// TwinCAT 3 PLC project SSP_M
// ProgramVersion: 3.1.4024.0
// libraries:
//   EfficientIO Communicator, * (EfficientIO)
//   EfficientIO Energy Basic, * (EfficientIO)
//   Lynus Persistent Data V1, * (Lynus AG)
//   Lynus Standards, * (EfficientIO)
//   Tc2_EtherCAT, * (Beckhoff Automation GmbH)
//   Tc2_Standard, * (Beckhoff Automation GmbH)
//   Tc2_System, * (Beckhoff Automation GmbH)
//   Tc2_Utilities, * (Beckhoff Automation GmbH)
//   Tc3_IPCDiag, * (Beckhoff Automation GmbH)
//   Tc3_Module, * (Beckhoff Automation GmbH)
// project tree:
//   ENUM/ E_State.TcDUT (not stored)
//   / FastTask.TcTTO, MiddleTask.TcTTO, SlowTask.TcTTO
//   FBs/EL3443_DPM/DUTs/ E_EL3443_DPM_Phase.TcDUT (not stored), E_EL3443_DPM_Total.TcDUT (not stored), MDP5001_341_7CD731EE.TcDUT (not stored), MDP5001_341_I_7CD731EE.TcDUT, MDP5001_341_O_7CD731EE.TcDUT (not stored), ST_EL3443_DPM_MUX_REAL.TcDUT (not stored), ST_EL3443_DPM_MUX_ULINT.TcDUT (not stored), ST_EL3443_DPM_StatusLx.TcDUT (not stored), ST_EL3443_DPM_StatusTotal.TcDUT (not stored), ST_EL3443_DPM_VariantLx.TcDUT (not stored), ST_EL3443_DPM_VariantTotal.TcDUT (not stored), ST_EL3443_DPM_VariantValues.TcDUT (not stored)
//   FBs/EL3443_DPM/ FB_EL3443_DPM.TcPOU (not stored)
//   FBs/EL3446 FW02 or higher/DUTs/ E_EL3446_Phase.TcDUT (not stored), MDP5001_342_066CA8C6.TcDUT (not stored), MDP5001_342_I_066CA8C6.TcDUT (not stored), MDP5001_342_O_066CA8C6.TcDUT (not stored), ST_EL3446_MUX_REAL.TcDUT (not stored), ST_EL3446_MUX_ULINT.TcDUT (not stored), ST_EL3446_StatusIx.TcDUT (not stored), ST_EL3446_VariantIx.TcDUT (not stored), ST_EL3446_VariantValues.TcDUT (not stored)
//   FBs/EL3446 FW02 or higher/ FB_EL3446.TcPOU (not stored)
//   FBs/ FB_CoE_EL3443.TcPOU (not stored), FB_CoE_EL3446.TcPOU (not stored), FB_EM_Beckhoff_EL3443.TcPOU (not stored), FB_EM_Beckhoff_EL3446.TcPOU (not stored), prg_ReadDeviceName.TcPOU (not stored)
//   POUs/ prgComEffIO.TcPOU, prgEM.TcPOU, prgHW.TcPOU, prgPersistent.TcPOU (not stored), prgRWEffIO.TcPOU, prgVarEffIO.TcPOU

CONFIGURATION SSP_M
    RESOURCE PLC ON TwinCAT3
        TASK FastTask(INTERVAL := T#10ms, PRIORITY := 21);
        TASK MiddleTask(INTERVAL := T#10ms, PRIORITY := 22);
        TASK SlowTask(INTERVAL := T#10ms, PRIORITY := 23);
        PROGRAM prgVarEffIO WITH FastTask : prgVarEffIO;
        PROGRAM prgRWEffIO WITH FastTask : prgRWEffIO;
        PROGRAM prgPersistent WITH MiddleTask : prgPersistent;
        PROGRAM prgEM WITH MiddleTask : prgEM;
        PROGRAM prgHW WITH MiddleTask : prgHW;
        PROGRAM prgComEffIO WITH SlowTask : prgComEffIO;
    END_RESOURCE
END_CONFIGURATION

// ---- FBs/EL3443_DPM/DUTs/MDP5001_341_I_7CD731EE.TcDUT
TYPE MDP5001_341_I_7CD731EE :
STRUCT
	MDP5001_341_L1_Status_Voltage_Sign_Bit			: BIT;
	MDP5001_341_L1_Status_Overvoltage				: BIT;
	MDP5001_341_L1_Status_Overcurrent				: BIT;
	MDP5001_341_L1_Status_Inaccurate_Voltage		: BIT;
	MDP5001_341_L1_Status_Inaccurate_Current		: BIT;
	MDP5001_341_L1_Status_Voltage_Guard_Warning		: BIT;
	MDP5001_341_L1_Status_Voltage_Guard_Error		: BIT;
	MDP5001_341_L1_Status_Current_Guard_Warning		: BIT;
	MDP5001_341_L1_Status_Current_Guard_Error		: BIT;
	MDP5001_341_L1_Status_TxPDO_Toggle				: BIT;
	MDP5001_341_L1_Basic_Voltage					: REAL;
	MDP5001_341_L1_Basic_Current					: REAL;
	MDP5001_341_L1_Power_Active_Power				: REAL;
	MDP5001_341_L1_Power_Apparent_Power				: REAL;
	MDP5001_341_L1_Power_Reactive_Power				: REAL;
	MDP5001_341_L1_Power_Power_Factor				: REAL;
	MDP5001_341_L2_Status_Voltage_Sign_Bit			: BIT;
	MDP5001_341_L2_Status_Overvoltage				: BIT;
	MDP5001_341_L2_Status_Overcurrent				: BIT;
	MDP5001_341_L2_Status_Inaccurate_Voltage		: BIT;
	MDP5001_341_L2_Status_Inaccurate_Current		: BIT;
	MDP5001_341_L2_Status_Voltage_Guard_Warning		: BIT;
	MDP5001_341_L2_Status_Voltage_Guard_Error		: BIT;
	MDP5001_341_L2_Status_Current_Guard_Warning		: BIT;
	MDP5001_341_L2_Status_Current_Guard_Error		: BIT;
	MDP5001_341_L2_Status_TxPDO_Toggle				: BIT;
	MDP5001_341_L2_Basic_Voltage					: REAL;
	MDP5001_341_L2_Basic_Current					: REAL;
	MDP5001_341_L2_Power_Active_Power				: REAL;
	MDP5001_341_L2_Power_Apparent_Power				: REAL;
	MDP5001_341_L2_Power_Reactive_Power				: REAL;
	MDP5001_341_L2_Power_Power_Factor				: REAL;
	MDP5001_341_L3_Status_Voltage_Sign_Bit			: BIT;
	MDP5001_341_L3_Status_Overvoltage				: BIT;
	MDP5001_341_L3_Status_Overcurrent				: BIT;
	MDP5001_341_L3_Status_Inaccurate_Voltage		: BIT;
	MDP5001_341_L3_Status_Inaccurate_Current		: BIT;
	MDP5001_341_L3_Status_Voltage_Guard_Warning		: BIT;
	MDP5001_341_L3_Status_Voltage_Guard_Error		: BIT;
	MDP5001_341_L3_Status_Current_Guard_Warning		: BIT;
	MDP5001_341_L3_Status_Current_Guard_Error		: BIT;
	MDP5001_341_L3_Status_TxPDO_Toggle				: BIT;
	MDP5001_341_L3_Basic_Voltage					: REAL;
	MDP5001_341_L3_Basic_Current					: REAL;
	MDP5001_341_L3_Power_Active_Power				: REAL;
	MDP5001_341_L3_Power_Apparent_Power				: REAL;
	MDP5001_341_L3_Power_Reactive_Power				: REAL;
	MDP5001_341_L3_Power_Power_Factor				: REAL;	
	MDP5001_341_Total_Status_System_State					: BIT;
	MDP5001_341_Total_Status_Grid_Direction					: BIT;
	MDP5001_341_Total_Status_Frequency_Guard_Warning		: BIT;
	MDP5001_341_Total_Status_Frequency_Guard_Error			: BIT;
	MDP5001_341_Total_Status_Neutral_Current_Guard_Warning	: BIT;
	MDP5001_341_Total_Status_Neutral_Current_Guard_Error	: BIT;
	MDP5001_341_Total_Status_Active_Power_Guard_Warning		: BIT;
	MDP5001_341_Total_Status_Active_Power_Guard_Error		: BIT;
	MDP5001_341_Total_Status_Apparent_Power_Guard_Warning	: BIT;
	MDP5001_341_Total_Status_Apparent_Power_Guard_Error		: BIT;
	MDP5001_341_Total_Status_Power_Quality_Guard_Warning	: BIT;
	MDP5001_341_Total_Status_Power_Quality_Guard_Error		: BIT;
	MDP5001_341_Total_Status_TxPDO_State					: BIT;
	MDP5001_341_Total_Status_TxPDO_Toggle					: BIT;
	MDP5001_341_Total_Status_Power_Quality_Factor			: REAL;	
	MDP5001_341_Total_Basic_Frequency						: REAL;	
	MDP5001_341_Total_Basic_Power_Factor					: REAL;	
	MDP5001_341_Total_Basic_Calculated_Neutral_Line_Current	: REAL;	
	MDP5001_341_Total_Variant_Value_In_TxPDO_Toggle			: BIT;
	MDP5001_341_Total_Variant_Value_In_Index_1_REAL			: UINT;
	MDP5001_341_Total_Variant_Value_In_Value_1_REAL			: REAL;
	MDP5001_341_Total_Variant_Value_In_Index_2_REAL			: UINT;
	MDP5001_341_Total_Variant_Value_In_Value_2_REAL			: REAL;
	MDP5001_341_Total_Variant_Value_In_Index_3_REAL			: UINT;
	MDP5001_341_Total_Variant_Value_In_Value_3_REAL			: REAL;
	MDP5001_341_Total_Variant_Value_In_Index_4_ULINT		: UINT;
	MDP5001_341_Total_Variant_Value_In_Value_4_ULINT		: ULINT;
	MDP5001_341_DPM_Data_Data_1								: UDINT;
	MDP5001_341_DPM_Data_Data_2								: UDINT;
	MDP5001_341_DPM_Data_Data_3								: UDINT;
	MDP5001_341_DPM_Data_Data_4								: UDINT;
	MDP5001_341_DPM_Data_Data_5								: UDINT;
	MDP5001_341_DPM_Data_Data_6								: UDINT;
	MDP5001_341_DPM_Data_Data_7								: UDINT;
	MDP5001_341_DPM_Data_Data_8								: UDINT;
	MDP5001_341_DPM_Data_Data_9								: UDINT;
	MDP5001_341_DPM_Data_Data_10							: UDINT;
	MDP5001_341_DPM_Data_Data_11							: UDINT;
	MDP5001_341_DPM_Data_Data_12							: UDINT;
	MDP5001_341_DPM_Data_Data_13							: UDINT;
	MDP5001_341_DPM_Data_Data_14							: UDINT;
	MDP5001_341_DPM_Data_Data_15							: UDINT;
	MDP5001_341_DPM_Data_Data_16							: UDINT;
	MDP5001_341_DPM_Data_Data_17							: UDINT;
	MDP5001_341_DPM_Data_Data_18							: UDINT;
	MDP5001_341_DPM_Data_Data_19							: UDINT;
	MDP5001_341_DPM_Data_Data_20							: UDINT;
END_STRUCT
END_TYPE

// ---- POUs/prgVarEffIO.TcPOU
PROGRAM prgVarEffIO
VAR
	fbVar		: FB_VarInfo;
END_VAR

fbVar(
	bReadInfo:= , 
	eTMCFile:= eSelectTMCFile.eDontUseTMCFile, 
	eSavePositionTMCFile:= eSavePositionOnPLC.ePostionHardDisk, 
	udiCounterFoundVariables=> , 
	bError=> , 
	bBusy=> , 
	byProgress=> , 
	udiErrorCodeOut=> , 
	eErrorVarInfo_Out=> , 
	sVarWithError=> );

END_PROGRAM

// ---- POUs/prgRWEffIO.TcPOU
PROGRAM prgRWEffIO
VAR
	fbRW1		: FB_ReadWrite_V2;
	fbRW2		: FB_ReadWrite;
	fbRW3		: FB_ReadWrite;
END_VAR

fbRW1(	eUploadType := eSelectDataUploadType.e_Change_noIntervall,
		bBusy=> , 
		bError=> , 
		udiErrorCodeOut=> , 
		eErrorReadWrite_Out=> );
		
fbRW2();
		
fbRW3();

END_PROGRAM

// ---- POUs/prgEM.TcPOU
PROGRAM prgEM
VAR
 	fb_EL3443_EM0 		: FB_EM_Beckhoff_EL3443;
	fb_EL3446_1			: FB_EM_Beckhoff_EL3446;
	fb_EL3446_2			: FB_EM_Beckhoff_EL3446;
	fb_EL3446_3			: FB_EM_Beckhoff_EL3446;
	fb_EL3446_4			: FB_EM_Beckhoff_EL3446;
	
	//EM0 (CEE32 3phase Measurement, EL3443)
	lr_RealPower_EM0		: LREAL;					//{#lynus.ag#()}
	lr_ApparentPower_EM0	: LREAL;					//{#lynus.ag#()}
	lr_ReactivePower_EM0	: LREAL;					//{#lynus.ag#()}
	lr_Frequency_EM0		: LREAL;					//{#lynus.ag#()}
	lr_Voltage_EM0_L1N		: LREAL;					//{#lynus.ag#()}
	lr_Voltage_EM0_L2N		: LREAL;					//{#lynus.ag#()}
	lr_Voltage_EM0_L3N		: LREAL;					//{#lynus.ag#()}
	lr_Voltage_EM0_L1L2		: LREAL;					//{#lynus.ag#()}
	lr_Voltage_EM0_L2L3		: LREAL;					//{#lynus.ag#()}
	lr_Voltage_EM0_L3L1		: LREAL;					//{#lynus.ag#()}
 	lr_Current_EM0_L1		: LREAL;					//{#lynus.ag#()}
	lr_Current_EM0_L2		: LREAL;					//{#lynus.ag#()}
	lr_Current_EM0_L3		: LREAL;					//{#lynus.ag#()}
	
	//EM1, EL3446-1
	lrPower_EM1_1		: LREAL;						//{#lynus.ag#()}
	lrPower_EM1_2		: LREAL;						//{#lynus.ag#()}
	lrPower_EM1_3		: LREAL;						//{#lynus.ag#()}
	lrPower_EM1_4		: LREAL;						//{#lynus.ag#()}
	lrPower_EM1_5		: LREAL;						//{#lynus.ag#()}
	lrPower_EM1_6		: LREAL;						//{#lynus.ag#()}
	lrPower_EM1_3p1		: LREAL;						//{#lynus.ag#()}
	lrPower_EM1_3p2		: LREAL;						//{#lynus.ag#()}
	
	//EM2, EL3446-2
	lrPower_EM2_1		: LREAL;						//{#lynus.ag#()}
	lrPower_EM2_2		: LREAL;						//{#lynus.ag#()}
	lrPower_EM2_3		: LREAL;						//{#lynus.ag#()}
	lrPower_EM2_4		: LREAL;						//{#lynus.ag#()}
	lrPower_EM2_5		: LREAL;						//{#lynus.ag#()}
	lrPower_EM2_6		: LREAL;						//{#lynus.ag#()}
	lrPower_EM2_3p1		: LREAL;						//{#lynus.ag#()}
	lrPower_EM2_3p2		: LREAL;						//{#lynus.ag#()}
	
	//EM3, EL3446-3
	lrPower_EM3_1		: LREAL;						//{#lynus.ag#()}
	lrPower_EM3_2		: LREAL;						//{#lynus.ag#()}
	lrPower_EM3_3		: LREAL;						//{#lynus.ag#()}
	lrPower_EM3_4		: LREAL;						//{#lynus.ag#()}
	lrPower_EM3_5		: LREAL;						//{#lynus.ag#()}
	lrPower_EM3_6		: LREAL;						//{#lynus.ag#()}
	lrPower_EM3_3p1		: LREAL;						//{#lynus.ag#()}
	lrPower_EM3_3p2		: LREAL;						//{#lynus.ag#()}
	
	//EM3, EL3446-4
	lrPower_EM4_1		: LREAL;						//{#lynus.ag#()}
	lrPower_EM4_2		: LREAL;						//{#lynus.ag#()}
	lrPower_EM4_3		: LREAL;						//{#lynus.ag#()}
	lrPower_EM4_4		: LREAL;						//{#lynus.ag#()}
	lrPower_EM4_5		: LREAL;						//{#lynus.ag#()}
	lrPower_EM4_6		: LREAL;						//{#lynus.ag#()}
	lrPower_EM4_3p1		: LREAL;						//{#lynus.ag#()}
	lrPower_EM4_3p2		: LREAL;						//{#lynus.ag#()}

END_VAR

VAR_INPUT
	stEL3443_IO_1 						: MDP5001_341_7CD731EE;
	stEL3446_IO_1 						: MDP5001_342_066CA8C6; 
	stEL3446_IO_2 						: MDP5001_342_066CA8C6;	
	stEL3446_IO_3 						: MDP5001_342_066CA8C6;	
	stEL3446_IO_4 						: MDP5001_342_066CA8C6;	
END_VAR

VAR PERSISTENT
	uiCurrentTransformerRatio_EM0	:UINT:=32;
	
	lr_EnergyCounter_EM0	: LREAL;
	lr_EnergyCounter_EM1	: LREAL;
	
	ui_PhaseSelector_EM1_1 : UINT := 1;						//{#lynus.ag#()}
	ui_PhaseSelector_EM1_2 : UINT := 2;						//{#lynus.ag#()}
	ui_PhaseSelector_EM1_3 : UINT := 3;						//{#lynus.ag#()}
	ui_PhaseSelector_EM2_1 : UINT := 1;						//{#lynus.ag#()}
	ui_PhaseSelector_EM2_2 : UINT := 2;						//{#lynus.ag#()}
	ui_PhaseSelector_EM2_3 : UINT := 3;						//{#lynus.ag#()}
	ui_PhaseSelector_EM2_4 : UINT := 1;						//{#lynus.ag#()}
	ui_PhaseSelector_EM2_5 : UINT := 2;						//{#lynus.ag#()}
	ui_PhaseSelector_EM2_6 : UINT := 3;						//{#lynus.ag#()}
	ui_PhaseSelector_EM3_1 : UINT := 1;						//{#lynus.ag#()}
	ui_PhaseSelector_EM3_2 : UINT := 2;						//{#lynus.ag#()}
	ui_PhaseSelector_EM3_3 : UINT := 3;						//{#lynus.ag#()}
	ui_PhaseSelector_EM3_4 : UINT := 1;						//{#lynus.ag#()}
	ui_PhaseSelector_EM3_5 : UINT := 2;						//{#lynus.ag#()}
	ui_PhaseSelector_EM3_6 : UINT := 3;						//{#lynus.ag#()}
	ui_PhaseSelector_EM4_1 : UINT := 1;						//{#lynus.ag#()}
	ui_PhaseSelector_EM4_2 : UINT := 2;						//{#lynus.ag#()}
	ui_PhaseSelector_EM4_3 : UINT := 3;						//{#lynus.ag#()}
	ui_PhaseSelector_EM4_4 : UINT := 1;						//{#lynus.ag#()}
	ui_PhaseSelector_EM4_5 : UINT := 2;						//{#lynus.ag#()}
	ui_PhaseSelector_EM4_6 : UINT := 3;						//{#lynus.ag#()}
	
	uiCurrentTransformerRatio_EM1_1	: UINT := 300;				//{#lynus.ag#()}
	uiCurrentTransformerRatio_EM1_2	: UINT := 300;				//{#lynus.ag#()}
	uiCurrentTransformerRatio_EM1_3	: UINT := 300;				//{#lynus.ag#()}
	uiCurrentTransformerRatio_EM2_1	: UINT := 300;				//{#lynus.ag#()}
	uiCurrentTransformerRatio_EM2_2	: UINT := 300;				//{#lynus.ag#()}
	uiCurrentTransformerRatio_EM2_3	: UINT := 300;				//{#lynus.ag#()}
	uiCurrentTransformerRatio_EM2_4	: UINT := 300;				//{#lynus.ag#()}
	uiCurrentTransformerRatio_EM2_5	: UINT := 300;				//{#lynus.ag#()}
	uiCurrentTransformerRatio_EM2_6	: UINT := 300;				//{#lynus.ag#()}
	uiCurrentTransformerRatio_EM3_1	: UINT := 300;				//{#lynus.ag#()}
	uiCurrentTransformerRatio_EM3_2	: UINT := 300;				//{#lynus.ag#()}
	uiCurrentTransformerRatio_EM3_3	: UINT := 300;				//{#lynus.ag#()}
	uiCurrentTransformerRatio_EM3_4	: UINT := 300;				//{#lynus.ag#()}
	uiCurrentTransformerRatio_EM3_5	: UINT := 300;				//{#lynus.ag#()}
	uiCurrentTransformerRatio_EM3_6	: UINT := 300;				//{#lynus.ag#()}
	uiCurrentTransformerRatio_EM4_1	: UINT := 300;				//{#lynus.ag#()}
	uiCurrentTransformerRatio_EM4_2	: UINT := 300;				//{#lynus.ag#()}
	uiCurrentTransformerRatio_EM4_3	: UINT := 300;				//{#lynus.ag#()}
	uiCurrentTransformerRatio_EM4_4	: UINT := 300;				//{#lynus.ag#()}
	uiCurrentTransformerRatio_EM4_5	: UINT := 300;				//{#lynus.ag#()}
	uiCurrentTransformerRatio_EM4_6	: UINT := 300;				//{#lynus.ag#()}
	
	b_Invers_EM1_1	:	BOOL := FALSE;							//{#lynus.ag#()}
	b_Invers_EM1_2	:	BOOL := FALSE;							//{#lynus.ag#()}
	b_Invers_EM1_3	:	BOOL := FALSE;							//{#lynus.ag#()}
	b_Invers_EM2_1	:	BOOL := FALSE;							//{#lynus.ag#()}
	b_Invers_EM2_2	:	BOOL := FALSE;							//{#lynus.ag#()}
	b_Invers_EM2_3	:	BOOL := FALSE;							//{#lynus.ag#()}
	b_Invers_EM2_4	:	BOOL := FALSE;							//{#lynus.ag#()}
	b_Invers_EM2_5	:	BOOL := FALSE;							//{#lynus.ag#()}
	b_Invers_EM2_6	:	BOOL := FALSE;							//{#lynus.ag#()}
	b_Invers_EM3_1	:	BOOL := FALSE;							//{#lynus.ag#()}
	b_Invers_EM3_2	:	BOOL := FALSE;							//{#lynus.ag#()}
	b_Invers_EM3_3	:	BOOL := FALSE;							//{#lynus.ag#()}
	b_Invers_EM3_4	:	BOOL := FALSE;							//{#lynus.ag#()}
	b_Invers_EM3_5	:	BOOL := FALSE;							//{#lynus.ag#()}
	b_Invers_EM3_6	:	BOOL := FALSE;							//{#lynus.ag#()}
	b_Invers_EM4_1	:	BOOL := FALSE;							//{#lynus.ag#()}
	b_Invers_EM4_2	:	BOOL := FALSE;							//{#lynus.ag#()}
	b_Invers_EM4_3	:	BOOL := FALSE;							//{#lynus.ag#()}
	b_Invers_EM4_4	:	BOOL := FALSE;							//{#lynus.ag#()}
	b_Invers_EM4_5	:	BOOL := FALSE;							//{#lynus.ag#()}
	b_Invers_EM4_6	:	BOOL := FALSE;							//{#lynus.ag#()}
END_VAR

//EM0 (CEE32 3phase Measurement)
fb_EL3443_EM0(
	bEnable 	:= TRUE, 
	bInvers_CH1 := , 
	bInvers_CH2	:= , 
	bInvers_CH3	:= , 
	uiCurrentTransformerRatio:= uiCurrentTransformerRatio_EM0, 
	nSlaveAddr 	:= 1001,
	stEL3443_IO := ,
	pDpmData=> , 
	stDataEMPower=> , 
	stDataEMCounter=> , 
	stDataEMPowerRealTime=> , 
	stDataEMCounterRealTime=> );

fb_EL3443_EM0.stEL3443_IO.MDP5001_341_Input := stEL3443_IO_1.MDP5001_341_Input;
stEL3443_IO_1.MDP5001_341_Output	:= fb_EL3443_EM0.stEL3443_IO.MDP5001_341_Output;
 	
lr_RealPower_EM0 			:= fb_EL3443_EM0.stDataEMPower.lrPowerTotal; 	
lr_ApparentPower_EM0 		:= fb_EL3443_EM0.stDataEMPower.lrApparentPowerTotal;
lr_ReactivePower_EM0		:= fb_EL3443_EM0.stDataEMPower.lrReactivePowerTotal;
lr_Frequency_EM0			:= fb_EL3443_EM0.stDataEMPower.lrFrequency;
lr_Voltage_EM0_L1N			:= fb_EL3443_EM0.stDataEMPower.lrVoltageL1N;
lr_Voltage_EM0_L2N			:= fb_EL3443_EM0.stDataEMPower.lrVoltageL2N;
lr_Voltage_EM0_L3N			:= fb_EL3443_EM0.stDataEMPower.lrVoltageL3N;
lr_Voltage_EM0_L1L2			:= fb_EL3443_EM0.stDataEMPower.lrVoltageL1L2;
lr_Voltage_EM0_L2L3			:= fb_EL3443_EM0.stDataEMPower.lrVoltageL2L3;
lr_Voltage_EM0_L3L1			:= fb_EL3443_EM0.stDataEMPower.lrVoltageL3L1;
lr_EnergyCounter_EM0		:= fb_EL3443_EM0.stDataEMCounter.lrTotalCounterEnergy_Consumption;
lr_Current_EM0_L1			:= fb_EL3443_EM0.stDataEMPower.lrCurrentL1;
lr_Current_EM0_L2			:= fb_EL3443_EM0.stDataEMPower.lrCurrentL2;
lr_Current_EM0_L3			:= fb_EL3443_EM0.stDataEMPower.lrCurrentL3;


//EM1 (for single Phase Measurements, EL3446-1)
fb_EL3446_1(
	bEnable:= TRUE , 
	bEnableVariantValues:= TRUE, 
	pDpmData:= fb_EL3443_EM0.pDpmData, 
	nSlaveAddr:= 1002, 
	bInvers_CH1:= b_Invers_EM2_1, 
	bInvers_CH2:= b_Invers_EM2_2, 
	bInvers_CH3:= b_Invers_EM2_3, 
	bInvers_CH4:= b_Invers_EM2_4, 
	bInvers_CH5:= b_Invers_EM2_5, 
	bInvers_CH6:= b_Invers_EM2_6, 
	uiCurrentTransformerRatio_CH1:= uiCurrentTransformerRatio_EM2_1, 
	uiCurrentTransformerRatio_CH2:= uiCurrentTransformerRatio_EM2_2, 
	uiCurrentTransformerRatio_CH3:= uiCurrentTransformerRatio_EM2_3, 
	uiCurrentTransformerRatio_CH4:= uiCurrentTransformerRatio_EM2_4, 
	uiCurrentTransformerRatio_CH5:= uiCurrentTransformerRatio_EM2_5, 
	uiCurrentTransformerRatio_CH6:= uiCurrentTransformerRatio_EM2_6, 
	uiVoltagePhaseSelector_CH1:= ui_PhaseSelector_EM2_1, 
	uiVoltagePhaseSelector_CH2:= ui_PhaseSelector_EM2_2, 
	uiVoltagePhaseSelector_CH3:= ui_PhaseSelector_EM2_3, 
	uiVoltagePhaseSelector_CH4:= ui_PhaseSelector_EM2_4, 
	uiVoltagePhaseSelector_CH5:= ui_PhaseSelector_EM2_5, 
	uiVoltagePhaseSelector_CH6:= ui_PhaseSelector_EM2_6, 
	bEnable3PhaseCH13:= FALSE, 
	bEnable3PhaseCH46:= FALSE, 
	stDataEMPowerRealTime:= fb_EL3443_EM0.stDataEMPowerRealTime, 
	stEL3446_IO := ,
	stDataEMPower_CH1=> , 
	stDataEMCounter_CH1=> , 
	stDataEMPowerRealTime_CH1=> , 
	stDataEMCounterRealTime_CH1=> , 
	stDataEMPower_CH2=> , 
	stDataEMCounter_CH2=> , 
	stDataEMPowerRealTime_CH2=> , 
	stDataEMCounterRealTime_CH2=> , 
	stDataEMPower_CH3=> , 
	stDataEMCounter_CH3=> , 
	stDataEMPowerRealTime_CH3=> , 
	stDataEMCounterRealTime_CH3=> , 
	stDataEMPower_CH4=> , 
	stDataEMCounter_CH4=> , 
	stDataEMPowerRealTime_CH4=> , 
	stDataEMCounterRealTime_CH4=> , 
	stDataEMPower_CH5=> , 
	stDataEMCounter_CH5=> , 
	stDataEMPowerRealTime_CH5=> , 
	stDataEMCounterRealTime_CH5=> , 
	stDataEMPower_CH6=> , 
	stDataEMCounter_CH6=> , 
	stDataEMPowerRealTime_CH6=> , 
	stDataEMCounterRealTime_CH6=> );
fb_EL3446_1.stEL3446_IO.MDP5001_342_Input := stEL3446_IO_1.MDP5001_342_Input;
stEL3446_IO_1.MDP5001_342_Output := 	fb_EL3446_1.stEL3446_IO.MDP5001_342_Output;

lrPower_EM2_1				:= 	LIMIT(0,fb_EL3446_1.stDataEMPower_CH1.lrPowerTotal,1000);
lrPower_EM2_2				:= 	LIMIT(0,fb_EL3446_1.stDataEMPower_CH2.lrPowerTotal,1000);
lrPower_EM2_3				:= 	LIMIT(0,fb_EL3446_1.stDataEMPower_CH3.lrPowerTotal,1000);
lrPower_EM2_4				:= 	LIMIT(0,fb_EL3446_1.stDataEMPower_CH4.lrPowerTotal,1000);
lrPower_EM2_5				:= 	LIMIT(0,fb_EL3446_1.stDataEMPower_CH5.lrPowerTotal,1000);
lrPower_EM2_6				:= 	LIMIT(0,fb_EL3446_1.stDataEMPower_CH6.lrPowerTotal,1000);

lrPower_EM2_3p1 			:= lrPower_EM2_1 + lrPower_EM2_2 + lrPower_EM2_3;
lrPower_EM2_3p2 			:= lrPower_EM2_4 + lrPower_EM2_5 + lrPower_EM2_6;

//EM2 (for single Phase Measurements, EL3446-2)
fb_EL3446_2(
	bEnable:= TRUE , 
	bEnableVariantValues:= TRUE, 
	pDpmData:= fb_EL3443_EM0.pDpmData, 
	nSlaveAddr:= 1003, 
	bInvers_CH1:= b_Invers_EM2_1, 
	bInvers_CH2:= b_Invers_EM2_2, 
	bInvers_CH3:= b_Invers_EM2_3, 
	bInvers_CH4:= b_Invers_EM2_4, 
	bInvers_CH5:= b_Invers_EM2_5, 
	bInvers_CH6:= b_Invers_EM2_6, 
	uiCurrentTransformerRatio_CH1:= uiCurrentTransformerRatio_EM2_1, 
	uiCurrentTransformerRatio_CH2:= uiCurrentTransformerRatio_EM2_2, 
	uiCurrentTransformerRatio_CH3:= uiCurrentTransformerRatio_EM2_3, 
	uiCurrentTransformerRatio_CH4:= uiCurrentTransformerRatio_EM2_4, 
	uiCurrentTransformerRatio_CH5:= uiCurrentTransformerRatio_EM2_5, 
	uiCurrentTransformerRatio_CH6:= uiCurrentTransformerRatio_EM2_6, 
	uiVoltagePhaseSelector_CH1:= ui_PhaseSelector_EM2_1, 
	uiVoltagePhaseSelector_CH2:= ui_PhaseSelector_EM2_2, 
	uiVoltagePhaseSelector_CH3:= ui_PhaseSelector_EM2_3, 
	uiVoltagePhaseSelector_CH4:= ui_PhaseSelector_EM2_4, 
	uiVoltagePhaseSelector_CH5:= ui_PhaseSelector_EM2_5, 
	uiVoltagePhaseSelector_CH6:= ui_PhaseSelector_EM2_6, 
	bEnable3PhaseCH13:= FALSE, 
	bEnable3PhaseCH46:= FALSE, 
	stDataEMPowerRealTime:= fb_EL3443_EM0.stDataEMPowerRealTime, 
	stEL3446_IO := ,
	stDataEMPower_CH1=> , 
	stDataEMCounter_CH1=> , 
	stDataEMPowerRealTime_CH1=> , 
	stDataEMCounterRealTime_CH1=> , 
	stDataEMPower_CH2=> , 
	stDataEMCounter_CH2=> , 
	stDataEMPowerRealTime_CH2=> , 
	stDataEMCounterRealTime_CH2=> , 
	stDataEMPower_CH3=> , 
	stDataEMCounter_CH3=> , 
	stDataEMPowerRealTime_CH3=> , 
	stDataEMCounterRealTime_CH3=> , 
	stDataEMPower_CH4=> , 
	stDataEMCounter_CH4=> , 
	stDataEMPowerRealTime_CH4=> , 
	stDataEMCounterRealTime_CH4=> , 
	stDataEMPower_CH5=> , 
	stDataEMCounter_CH5=> , 
	stDataEMPowerRealTime_CH5=> , 
	stDataEMCounterRealTime_CH5=> , 
	stDataEMPower_CH6=> , 
	stDataEMCounter_CH6=> , 
	stDataEMPowerRealTime_CH6=> , 
	stDataEMCounterRealTime_CH6=> );
fb_EL3446_1.stEL3446_IO.MDP5001_342_Input := stEL3446_IO_1.MDP5001_342_Input;
stEL3446_IO_1.MDP5001_342_Output := 	fb_EL3446_1.stEL3446_IO.MDP5001_342_Output;

lrPower_EM2_1				:= 	LIMIT(0,fb_EL3446_1.stDataEMPower_CH1.lrPowerTotal,1000);
lrPower_EM2_2				:= 	LIMIT(0,fb_EL3446_1.stDataEMPower_CH2.lrPowerTotal,1000);
lrPower_EM2_3				:= 	LIMIT(0,fb_EL3446_1.stDataEMPower_CH3.lrPowerTotal,1000);
lrPower_EM2_4				:= 	LIMIT(0,fb_EL3446_1.stDataEMPower_CH4.lrPowerTotal,1000);
lrPower_EM2_5				:= 	LIMIT(0,fb_EL3446_1.stDataEMPower_CH5.lrPowerTotal,1000);
lrPower_EM2_6				:= 	LIMIT(0,fb_EL3446_1.stDataEMPower_CH6.lrPowerTotal,1000);

lrPower_EM2_3p1 			:= lrPower_EM2_1 + lrPower_EM2_2 + lrPower_EM2_3;
lrPower_EM2_3p2 			:= lrPower_EM2_4 + lrPower_EM2_5 + lrPower_EM2_6;

(*
lr_EnergyCounter_EM1	:= 	fb_EL3446_1.stDataEMCounter_CH1.lrTotalCounterEnergy_Consumption;
lr_EnergyCounter_EM2	:= 	fb_EL3446_1.stDataEMCounter_CH2.lrTotalCounterEnergy_Consumption;
lr_EnergyCounter_EM3	:= 	fb_EL3446_1.stDataEMCounter_CH3.lrTotalCounterEnergy_Consumption;
lr_EnergyCounter_EM4	:= 	fb_EL3446_1.stDataEMCounter_CH4.lrTotalCounterEnergy_Consumption;
lr_EnergyCounter_EM5	:= 	fb_EL3446_1.stDataEMCounter_CH5.lrTotalCounterEnergy_Consumption;
lr_EnergyCounter_EM6	:= 	fb_EL3446_1.stDataEMCounter_CH6.lrTotalCounterEnergy_Consumption;
*)

//EM3 (for single Phase Measurements, EL3446-3)
fb_EL3446_3(
	bEnable:= TRUE , 
	bEnableVariantValues:= TRUE, 
	pDpmData:= fb_EL3443_EM0.pDpmData, 
	nSlaveAddr:= 1004, 
	bInvers_CH1:= b_Invers_EM3_1, 
	bInvers_CH2:= b_Invers_EM3_2, 
	bInvers_CH3:= b_Invers_EM3_3, 
	bInvers_CH4:= b_Invers_EM3_4, 
	bInvers_CH5:= b_Invers_EM3_5, 
	bInvers_CH6:= b_Invers_EM3_6, 
	uiCurrentTransformerRatio_CH1:= uiCurrentTransformerRatio_EM3_1, 
	uiCurrentTransformerRatio_CH2:= uiCurrentTransformerRatio_EM3_2, 
	uiCurrentTransformerRatio_CH3:= uiCurrentTransformerRatio_EM3_3, 
	uiCurrentTransformerRatio_CH4:= uiCurrentTransformerRatio_EM3_4, 
	uiCurrentTransformerRatio_CH5:= uiCurrentTransformerRatio_EM3_5, 
	uiCurrentTransformerRatio_CH6:= uiCurrentTransformerRatio_EM3_6, 
	uiVoltagePhaseSelector_CH1:= ui_PhaseSelector_EM3_1, 
	uiVoltagePhaseSelector_CH2:= ui_PhaseSelector_EM3_2, 
	uiVoltagePhaseSelector_CH3:= ui_PhaseSelector_EM3_3, 
	uiVoltagePhaseSelector_CH4:= ui_PhaseSelector_EM3_4, 
	uiVoltagePhaseSelector_CH5:= ui_PhaseSelector_EM3_5, 
	uiVoltagePhaseSelector_CH6:= ui_PhaseSelector_EM3_6, 
	bEnable3PhaseCH13:= FALSE, 
	bEnable3PhaseCH46:= FALSE, 
	stDataEMPowerRealTime:= fb_EL3443_EM0.stDataEMPowerRealTime, 
	stEL3446_IO := ,
	stDataEMPower_CH1=> , 
	stDataEMCounter_CH1=> , 
	stDataEMPowerRealTime_CH1=> , 
	stDataEMCounterRealTime_CH1=> , 
	stDataEMPower_CH2=> , 
	stDataEMCounter_CH2=> , 
	stDataEMPowerRealTime_CH2=> , 
	stDataEMCounterRealTime_CH2=> , 
	stDataEMPower_CH3=> , 
	stDataEMCounter_CH3=> , 
	stDataEMPowerRealTime_CH3=> , 
	stDataEMCounterRealTime_CH3=> , 
	stDataEMPower_CH4=> , 
	stDataEMCounter_CH4=> , 
	stDataEMPowerRealTime_CH4=> , 
	stDataEMCounterRealTime_CH4=> , 
	stDataEMPower_CH5=> , 
	stDataEMCounter_CH5=> , 
	stDataEMPowerRealTime_CH5=> , 
	stDataEMCounterRealTime_CH5=> , 
	stDataEMPower_CH6=> , 
	stDataEMCounter_CH6=> , 
	stDataEMPowerRealTime_CH6=> , 
	stDataEMCounterRealTime_CH6=> );
fb_EL3446_2.stEL3446_IO.MDP5001_342_Input := stEL3446_IO_2.MDP5001_342_Input;
stEL3446_IO_2.MDP5001_342_Output := 	fb_EL3446_2.stEL3446_IO.MDP5001_342_Output;

lrPower_EM3_1				:= 	LIMIT(0,fb_EL3446_2.stDataEMPower_CH1.lrPowerTotal,1000);
lrPower_EM3_2				:= 	LIMIT(0,fb_EL3446_2.stDataEMPower_CH2.lrPowerTotal,1000);
lrPower_EM3_3				:= 	LIMIT(0,fb_EL3446_2.stDataEMPower_CH3.lrPowerTotal,1000);
lrPower_EM3_4				:= 	LIMIT(0,fb_EL3446_2.stDataEMPower_CH4.lrPowerTotal,1000);
lrPower_EM3_5				:= 	LIMIT(0,fb_EL3446_2.stDataEMPower_CH5.lrPowerTotal,1000);
lrPower_EM3_6				:= 	LIMIT(0,fb_EL3446_2.stDataEMPower_CH6.lrPowerTotal,1000);

lrPower_EM3_3p1 			:= lrPower_EM3_1 + lrPower_EM3_2 + lrPower_EM3_3;
lrPower_EM3_3p2 			:= lrPower_EM3_4 + lrPower_EM3_5 + lrPower_EM3_6;


//EM4 (for single Phase Measurements, EL3446-4)
fb_EL3446_4(
	bEnable:= TRUE , 
	bEnableVariantValues:= TRUE, 
	pDpmData:= fb_EL3443_EM0.pDpmData, 
	nSlaveAddr:= 1005, 
	bInvers_CH1:= b_Invers_EM4_1, 
	bInvers_CH2:= b_Invers_EM4_2, 
	bInvers_CH3:= b_Invers_EM4_3, 
	bInvers_CH4:= b_Invers_EM4_4, 
	bInvers_CH5:= b_Invers_EM4_5, 
	bInvers_CH6:= b_Invers_EM4_6, 
	uiCurrentTransformerRatio_CH1:= uiCurrentTransformerRatio_EM4_1, 
	uiCurrentTransformerRatio_CH2:= uiCurrentTransformerRatio_EM4_2, 
	uiCurrentTransformerRatio_CH3:= uiCurrentTransformerRatio_EM4_3, 
	uiCurrentTransformerRatio_CH4:= uiCurrentTransformerRatio_EM4_4, 
	uiCurrentTransformerRatio_CH5:= uiCurrentTransformerRatio_EM4_5, 
	uiCurrentTransformerRatio_CH6:= uiCurrentTransformerRatio_EM4_6, 
	uiVoltagePhaseSelector_CH1:= ui_PhaseSelector_EM4_1, 
	uiVoltagePhaseSelector_CH2:= ui_PhaseSelector_EM4_2, 
	uiVoltagePhaseSelector_CH3:= ui_PhaseSelector_EM4_3, 
	uiVoltagePhaseSelector_CH4:= ui_PhaseSelector_EM4_4, 
	uiVoltagePhaseSelector_CH5:= ui_PhaseSelector_EM4_5, 
	uiVoltagePhaseSelector_CH6:= ui_PhaseSelector_EM4_6, 
	bEnable3PhaseCH13:= FALSE, 
	bEnable3PhaseCH46:= FALSE, 
	stDataEMPowerRealTime:= fb_EL3443_EM0.stDataEMPowerRealTime, 
	stEL3446_IO := ,
	stDataEMPower_CH1=> , 
	stDataEMCounter_CH1=> , 
	stDataEMPowerRealTime_CH1=> , 
	stDataEMCounterRealTime_CH1=> , 
	stDataEMPower_CH2=> , 
	stDataEMCounter_CH2=> , 
	stDataEMPowerRealTime_CH2=> , 
	stDataEMCounterRealTime_CH2=> , 
	stDataEMPower_CH3=> , 
	stDataEMCounter_CH3=> , 
	stDataEMPowerRealTime_CH3=> , 
	stDataEMCounterRealTime_CH3=> , 
	stDataEMPower_CH4=> , 
	stDataEMCounter_CH4=> , 
	stDataEMPowerRealTime_CH4=> , 
	stDataEMCounterRealTime_CH4=> , 
	stDataEMPower_CH5=> , 
	stDataEMCounter_CH5=> , 
	stDataEMPowerRealTime_CH5=> , 
	stDataEMCounterRealTime_CH5=> , 
	stDataEMPower_CH6=> , 
	stDataEMCounter_CH6=> , 
	stDataEMPowerRealTime_CH6=> , 
	stDataEMCounterRealTime_CH6=> );
fb_EL3446_2.stEL3446_IO.MDP5001_342_Input := stEL3446_IO_2.MDP5001_342_Input;
stEL3446_IO_2.MDP5001_342_Output := 	fb_EL3446_2.stEL3446_IO.MDP5001_342_Output;

lrPower_EM4_1				:= 	LIMIT(0,fb_EL3446_2.stDataEMPower_CH1.lrPowerTotal,1000);
lrPower_EM4_2				:= 	LIMIT(0,fb_EL3446_2.stDataEMPower_CH2.lrPowerTotal,1000);
lrPower_EM4_3				:= 	LIMIT(0,fb_EL3446_2.stDataEMPower_CH3.lrPowerTotal,1000);
lrPower_EM4_4				:= 	LIMIT(0,fb_EL3446_2.stDataEMPower_CH4.lrPowerTotal,1000);
lrPower_EM4_5				:= 	LIMIT(0,fb_EL3446_2.stDataEMPower_CH5.lrPowerTotal,1000);
lrPower_EM4_6				:= 	LIMIT(0,fb_EL3446_2.stDataEMPower_CH6.lrPowerTotal,1000);

lrPower_EM4_3p1 			:= lrPower_EM4_1 + lrPower_EM4_2 + lrPower_EM4_3;
lrPower_EM4_3p2 			:= lrPower_EM4_4 + lrPower_EM4_5 + lrPower_EM4_6;

END_PROGRAM

// ---- POUs/prgHW.TcPOU
PROGRAM prgHW
VAR

	// IOs for EL3443
	{attribute 'TcLinkTo' := 'TIID^Device 2 (EtherCAT)^Term 1 (EK1200)^Term 2 (EL3443)^L1 Status^Voltage Sign Bit'}
	MDP5001_341_L1_Status_Voltage_Sign_Bit   	AT%I*  : BOOL;  // linked via attribute 
	{attribute 'TcLinkTo' := 'TIID^Device 2 (EtherCAT)^Term 1 (EK1200)^Term 2 (EL3443)^L1 Status^Overvoltage'}
	MDP5001_341_L1_Status_Overvoltage			AT%I*  : BOOL;  // linked via attribute 
	{attribute 'TcLinkTo' := 'TIID^Device 2 (EtherCAT)^Term 1 (EK1200)^Term 2 (EL3443)^L1 Status^Overcurrent'}
	MDP5001_341_L1_Status_Overcurrent			AT%I*  : BOOL;  // linked via attribute 
	{attribute 'TcLinkTo' := 'TIID^Device 2 (EtherCAT)^Term 1 (EK1200)^Term 2 (EL3443)^L1 Status^Inaccurate Voltage'}	
	MDP5001_341_L1_Status_Inaccurate_Voltage	AT%I*  : BOOL;  // linked via attribute 
	{attribute 'TcLinkTo' := 'TIID^Device 2 (EtherCAT)^Term 1 (EK1200)^Term 2 (EL3443)^L1 Status^Inaccurate Current'}
	MDP5001_341_L1_Status_Inaccurate_Current	AT%I*  : BOOL;  // linked via attribute 	
	{attribute 'TcLinkTo' := 'TIID^Device 2 (EtherCAT)^Term 1 (EK1200)^Term 2 (EL3443)^L1 Status^Voltage Guard Warning'}
	MDP5001_341_L1_Status_Voltage_Guard_Warning	AT%I*  : BOOL;  // linked via attribute
	{attribute 'TcLinkTo' := 'TIID^Device 2 (EtherCAT)^Term 1 (EK1200)^Term 2 (EL3443)^L1 Status^Voltage Guard Error'}
	MDP5001_341_L1_Status_Voltage_Guard_Error	AT%I*  : BOOL;  // linked via attribute
	{attribute 'TcLinkTo' := 'TIID^Device 2 (EtherCAT)^Term 1 (EK1200)^Term 2 (EL3443)^L1 Status^Current Guard Warning'}
	MDP5001_341_L1_Status_Current_Guard_Warning AT%I*  : BOOL;  // linked via attribute
	{attribute 'TcLinkTo' := 'TIID^Device 2 (EtherCAT)^Term 1 (EK1200)^Term 2 (EL3443)^L1 Status^Current Guard Error'}
	MDP5001_341_L1_Status_Current_Guard_Error	AT%I*  : BOOL;  // linked via attribute
	{attribute 'TcLinkTo' := 'TIID^Device 2 (EtherCAT)^Term 1 (EK1200)^Term 2 (EL3443)^L1 Status^TxPDO Toggle'}
	MDP5001_341_L1_Status_TxPDO_Toggle			AT%I*  : BOOL;  // linked via attribute
	{attribute 'TcLinkTo' := 'TIID^Device 2 (EtherCAT)^Term 1 (EK1200)^Term 2 (EL3443)^L1 Basic^Voltage'}
	MDP5001_341_L1_Basic_Voltage				AT%I*  : REAL;		// linked via attribute 
	{attribute 'TcLinkTo' := 'TIID^Device 2 (EtherCAT)^Term 1 (EK1200)^Term 2 (EL3443)^L1 Basic^Current'}
	MDP5001_341_L1_Basic_Current				AT%I*  : REAL;		// linked via attribute 
	{attribute 'TcLinkTo' := 'TIID^Device 2 (EtherCAT)^Term 1 (EK1200)^Term 2 (EL3443)^L1 Power^Active Power'}
	MDP5001_341_L1_Power_Active_Power			AT%I*  : REAL;		// linked via attribute 
	{attribute 'TcLinkTo' := 'TIID^Device 2 (EtherCAT)^Term 1 (EK1200)^Term 2 (EL3443)^L1 Power^Apparent Power'}
	MDP5001_341_L1_Power_Apparent_Power			AT%I* : REAL;		// linked via attribute 
	{attribute 'TcLinkTo' := 'TIID^Device 2 (EtherCAT)^Term 1 (EK1200)^Term 2 (EL3443)^L1 Power^Reactive Power'}
	MDP5001_341_L1_Power_Reactive_Power			AT%I* : REAL;		// linked via attribute 
	{attribute 'TcLinkTo' := 'TIID^Device 2 (EtherCAT)^Term 1 (EK1200)^Term 2 (EL3443)^L1 Power^Power Factor'}
	MDP5001_341_L1_Power_Power_Factor			AT%I* : REAL;		// linked via attribute 
	{attribute 'TcLinkTo' := 'TIID^Device 2 (EtherCAT)^Term 1 (EK1200)^Term 2 (EL3443)^L2 Status^Voltage Sign Bit'}
	MDP5001_341_L2_Status_Voltage_Sign_Bit   	AT%I*  : BOOL;  // linked via attribute 
	{attribute 'TcLinkTo' := 'TIID^Device 2 (EtherCAT)^Term 1 (EK1200)^Term 2 (EL3443)^L2 Status^Overvoltage'}
	MDP5001_341_L2_Status_Overvoltage			AT%I*  : BOOL;  // linked via attribute 
	{attribute 'TcLinkTo' := 'TIID^Device 2 (EtherCAT)^Term 1 (EK1200)^Term 2 (EL3443)^L2 Status^Overcurrent'}
	MDP5001_341_L2_Status_Overcurrent			AT%I*  : BOOL;  // linked via attribute 
	{attribute 'TcLinkTo' := 'TIID^Device 2 (EtherCAT)^Term 1 (EK1200)^Term 2 (EL3443)^L2 Status^Inaccurate Voltage'}	
	MDP5001_341_L2_Status_Inaccurate_Voltage	AT%I*  : BOOL;  // linked via attribute 
	{attribute 'TcLinkTo' := 'TIID^Device 2 (EtherCAT)^Term 1 (EK1200)^Term 2 (EL3443)^L2 Status^Inaccurate Current'}
	MDP5001_341_L2_Status_Inaccurate_Current	AT%I*  : BOOL;  // linked via attribute 	
	{attribute 'TcLinkTo' := 'TIID^Device 2 (EtherCAT)^Term 1 (EK1200)^Term 2 (EL3443)^L2 Status^Voltage Guard Warning'}
	MDP5001_341_L2_Status_Voltage_Guard_Warning	AT%I*  : BOOL;  // linked via attribute
	{attribute 'TcLinkTo' := 'TIID^Device 2 (EtherCAT)^Term 1 (EK1200)^Term 2 (EL3443)^L2 Status^Voltage Guard Error'}
	MDP5001_341_L2_Status_Voltage_Guard_Error	AT%I*  : BOOL;  // linked via attribute
	{attribute 'TcLinkTo' := 'TIID^Device 2 (EtherCAT)^Term 1 (EK1200)^Term 2 (EL3443)^L2 Status^Current Guard Warning'}
	MDP5001_341_L2_Status_Current_Guard_Warning AT%I*  : BOOL;  // linked via attribute
	{attribute 'TcLinkTo' := 'TIID^Device 2 (EtherCAT)^Term 1 (EK1200)^Term 2 (EL3443)^L2 Status^Current Guard Error'}
	MDP5001_341_L2_Status_Current_Guard_Error	AT%I*  : BOOL;  // linked via attribute
	{attribute 'TcLinkTo' := 'TIID^Device 2 (EtherCAT)^Term 1 (EK1200)^Term 2 (EL3443)^L2 Status^TxPDO Toggle'}
	MDP5001_341_L2_Status_TxPDO_Toggle			AT%I*  : BOOL;  // linked via attribute
	{attribute 'TcLinkTo' := 'TIID^Device 2 (EtherCAT)^Term 1 (EK1200)^Term 2 (EL3443)^L2 Basic^Voltage'}
	MDP5001_341_L2_Basic_Voltage				AT%I* : REAL;		// linked via attribute 
	{attribute 'TcLinkTo' := 'TIID^Device 2 (EtherCAT)^Term 1 (EK1200)^Term 2 (EL3443)^L2 Basic^Current'}
	MDP5001_341_L2_Basic_Current				AT%I* : REAL;		// linked via attribute 
	{attribute 'TcLinkTo' := 'TIID^Device 2 (EtherCAT)^Term 1 (EK1200)^Term 2 (EL3443)^L2 Power^Active Power'}
	MDP5001_341_L2_Power_Active_Power			AT%I* : REAL;		// linked via attribute 
	{attribute 'TcLinkTo' := 'TIID^Device 2 (EtherCAT)^Term 1 (EK1200)^Term 2 (EL3443)^L2 Power^Apparent Power'}
	MDP5001_341_L2_Power_Apparent_Power			AT%I* : REAL;		// linked via attribute 
	{attribute 'TcLinkTo' := 'TIID^Device 2 (EtherCAT)^Term 1 (EK1200)^Term 2 (EL3443)^L2 Power^Reactive Power'}
	MDP5001_341_L2_Power_Reactive_Power			AT%I* : REAL;		// linked via attribute 
	{attribute 'TcLinkTo' := 'TIID^Device 2 (EtherCAT)^Term 1 (EK1200)^Term 2 (EL3443)^L2 Power^Power Factor'}
	MDP5001_341_L2_Power_Power_Factor			AT%I* : REAL;		// linked via attribute 
	{attribute 'TcLinkTo' := 'TIID^Device 2 (EtherCAT)^Term 1 (EK1200)^Term 2 (EL3443)^L3 Status^Voltage Sign Bit'}
	MDP5001_341_L3_Status_Voltage_Sign_Bit   	AT%I*  : BOOL;  // linked via attribute 
	{attribute 'TcLinkTo' := 'TIID^Device 2 (EtherCAT)^Term 1 (EK1200)^Term 2 (EL3443)^L3 Status^Overvoltage'}
	MDP5001_341_L3_Status_Overvoltage			AT%I*  : BOOL;  // linked via attribute 
	{attribute 'TcLinkTo' := 'TIID^Device 2 (EtherCAT)^Term 1 (EK1200)^Term 2 (EL3443)^L3 Status^Overcurrent'}
	MDP5001_341_L3_Status_Overcurrent			AT%I*  : BOOL;  // linked via attribute 
	{attribute 'TcLinkTo' := 'TIID^Device 2 (EtherCAT)^Term 1 (EK1200)^Term 2 (EL3443)^L3 Status^Inaccurate Voltage'}	
	MDP5001_341_L3_Status_Inaccurate_Voltage	AT%I*  : BOOL;  // linked via attribute 
	{attribute 'TcLinkTo' := 'TIID^Device 2 (EtherCAT)^Term 1 (EK1200)^Term 2 (EL3443)^L3 Status^Inaccurate Current'}
	MDP5001_341_L3_Status_Inaccurate_Current	AT%I*  : BOOL;  // linked via attribute 	
	{attribute 'TcLinkTo' := 'TIID^Device 2 (EtherCAT)^Term 1 (EK1200)^Term 2 (EL3443)^L3 Status^Voltage Guard Warning'}
	MDP5001_341_L3_Status_Voltage_Guard_Warning	AT%I*  : BOOL;  // linked via attribute
	{attribute 'TcLinkTo' := 'TIID^Device 2 (EtherCAT)^Term 1 (EK1200)^Term 2 (EL3443)^L3 Status^Voltage Guard Error'}
	MDP5001_341_L3_Status_Voltage_Guard_Error	AT%I*  : BOOL;  // linked via attribute
	{attribute 'TcLinkTo' := 'TIID^Device 2 (EtherCAT)^Term 1 (EK1200)^Term 2 (EL3443)^L3 Status^Current Guard Warning'}
	MDP5001_341_L3_Status_Current_Guard_Warning AT%I*  : BOOL;  // linked via attribute
	{attribute 'TcLinkTo' := 'TIID^Device 2 (EtherCAT)^Term 1 (EK1200)^Term 2 (EL3443)^L3 Status^Current Guard Error'}
	MDP5001_341_L3_Status_Current_Guard_Error	AT%I*  : BOOL;  // linked via attribute
	{attribute 'TcLinkTo' := 'TIID^Device 2 (EtherCAT)^Term 1 (EK1200)^Term 2 (EL3443)^L3 Status^TxPDO Toggle'}
	MDP5001_341_L3_Status_TxPDO_Toggle			AT%I*  : BOOL;  // linked via attribute
	{attribute 'TcLinkTo' := 'TIID^Device 2 (EtherCAT)^Term 1 (EK1200)^Term 2 (EL3443)^L3 Basic^Voltage'}
	MDP5001_341_L3_Basic_Voltage				AT%I* : REAL;		// linked via attribute 
	{attribute 'TcLinkTo' := 'TIID^Device 2 (EtherCAT)^Term 1 (EK1200)^Term 2 (EL3443)^L3 Basic^Current'}
	MDP5001_341_L3_Basic_Current				AT%I* : REAL;		// linked via attribute 
	{attribute 'TcLinkTo' := 'TIID^Device 2 (EtherCAT)^Term 1 (EK1200)^Term 2 (EL3443)^L3 Power^Active Power'}
	MDP5001_341_L3_Power_Active_Power			AT%I* : REAL;		// linked via attribute 
	{attribute 'TcLinkTo' := 'TIID^Device 2 (EtherCAT)^Term 1 (EK1200)^Term 2 (EL3443)^L3 Power^Apparent Power'}
	MDP5001_341_L3_Power_Apparent_Power			AT%I* : REAL;		// linked via attribute 
	{attribute 'TcLinkTo' := 'TIID^Device 2 (EtherCAT)^Term 1 (EK1200)^Term 2 (EL3443)^L3 Power^Reactive Power'}
	MDP5001_341_L3_Power_Reactive_Power			AT%I* : REAL;		// linked via attribute 
	{attribute 'TcLinkTo' := 'TIID^Device 2 (EtherCAT)^Term 1 (EK1200)^Term 2 (EL3443)^L3 Power^Power Factor'}
	MDP5001_341_L3_Power_Power_Factor			AT%I* : REAL;		// linked via attribute 
	{attribute 'TcLinkTo' := 'TIID^Device 2 (EtherCAT)^Term 1 (EK1200)^Term 2 (EL3443)^Total Status^System State'}
	MDP5001_341_Total_Status_System_State				AT%I* : BOOL;		// linked via attribute 
	{attribute 'TcLinkTo' := 'TIID^Device 2 (EtherCAT)^Term 1 (EK1200)^Term 2 (EL3443)^Total Status^Grid Direction'}
	MDP5001_341_Total_Status_Grid_Direction				AT%I* : BOOL;		// linked via attribute 
	{attribute 'TcLinkTo' := 'TIID^Device 2 (EtherCAT)^Term 1 (EK1200)^Term 2 (EL3443)^Total Status^Frequency Guard Warning'}
	MDP5001_341_Total_Status_Frequency_Guard_Warning	AT%I* : BOOL;		// linked via attribute 
	{attribute 'TcLinkTo' := 'TIID^Device 2 (EtherCAT)^Term 1 (EK1200)^Term 2 (EL3443)^Total Status^Frequency Guard Error'}
	MDP5001_341_Total_Status_Frequency_Guard_Error		AT%I* : BOOL;		// linked via attribute 
	{attribute 'TcLinkTo' := 'TIID^Device 2 (EtherCAT)^Term 1 (EK1200)^Term 2 (EL3443)^Total Status^Neutral Current Guard Warning'}
	MDP5001_341_Total_Status_Neutral_Current_Guard_Warning	AT%I* : BOOL;		// linked via attribute 
	{attribute 'TcLinkTo' := 'TIID^Device 2 (EtherCAT)^Term 1 (EK1200)^Term 2 (EL3443)^Total Status^Neutral Current Guard Error'}
	MDP5001_341_Total_Status_Neutral_Current_Guard_Error	AT%I* : BOOL;		// linked via attribute 
	{attribute 'TcLinkTo' := 'TIID^Device 2 (EtherCAT)^Term 1 (EK1200)^Term 2 (EL3443)^Total Status^Active Power Guard Warning'}
	MDP5001_341_Total_Status_Active_Power_Guard_Warning		AT%I* : BOOL;		// linked via attribute 
	{attribute 'TcLinkTo' := 'TIID^Device 2 (EtherCAT)^Term 1 (EK1200)^Term 2 (EL3443)^Total Status^Active Power Guard Error'}
	MDP5001_341_Total_Status_Active_Power_Guard_Error		AT%I* : BOOL;		// linked via attribute 
	{attribute 'TcLinkTo' := 'TIID^Device 2 (EtherCAT)^Term 1 (EK1200)^Term 2 (EL3443)^Total Status^Apparent Power Guard Warning'}
	MDP5001_341_Total_Status_Apparent_Power_Guard_Warning	AT%I* : BOOL;		// linked via attribute 
	{attribute 'TcLinkTo' := 'TIID^Device 2 (EtherCAT)^Term 1 (EK1200)^Term 2 (EL3443)^Total Status^Apparent Power Guard Error'}
	MDP5001_341_Total_Status_Apparent_Power_Guard_Error		AT%I* : BOOL;		// linked via attribute 
	{attribute 'TcLinkTo' := 'TIID^Device 2 (EtherCAT)^Term 1 (EK1200)^Term 2 (EL3443)^Total Status^Power Quality Guard Warning'}
	MDP5001_341_Total_Status_Power_Quality_Guard_Warning	AT%I* : BOOL;		// linked via attribute 
	{attribute 'TcLinkTo' := 'TIID^Device 2 (EtherCAT)^Term 1 (EK1200)^Term 2 (EL3443)^Total Status^Power Quality Guard Error'}
	MDP5001_341_Total_Status_Power_Quality_Guard_Error		AT%I* : BOOL;		// linked via attribute 
	{attribute 'TcLinkTo' := 'TIID^Device 2 (EtherCAT)^Term 1 (EK1200)^Term 2 (EL3443)^Total Status^TxPDO State'}
	MDP5001_341_Total_Status_TxPDO_State					AT%I* : BOOL;		// linked via attribute 
	{attribute 'TcLinkTo' := 'TIID^Device 2 (EtherCAT)^Term 1 (EK1200)^Term 2 (EL3443)^Total Status^TxPDO Toggle'}
	MDP5001_341_Total_Status_TxPDO_Toggle					AT%I* : BOOL;		// linked via attribute 
	{attribute 'TcLinkTo' := 'TIID^Device 2 (EtherCAT)^Term 1 (EK1200)^Term 2 (EL3443)^Total Status^Power Quality Factor'}
	MDP5001_341_Total_Status_Power_Quality_Factor			AT%I* : REAL;		// linked via attribute 
	{attribute 'TcLinkTo' := 'TIID^Device 2 (EtherCAT)^Term 1 (EK1200)^Term 2 (EL3443)^Total Basic^Frequency'}
	MDP5001_341_Total_Basic_Frequency						AT%I* : REAL;		// linked via attribute 
	{attribute 'TcLinkTo' := 'TIID^Device 2 (EtherCAT)^Term 1 (EK1200)^Term 2 (EL3443)^Total Basic^Power Factor'}
	MDP5001_341_Total_Basic_Power_Factor					AT%I* : REAL;		// linked via attribute 
	{attribute 'TcLinkTo' := 'TIID^Device 2 (EtherCAT)^Term 1 (EK1200)^Term 2 (EL3443)^Total Basic^Calculated Neutral Line Current'}
	MDP5001_341_Total_Basic_Calculated_Neutral_Line_Current	AT%I* : REAL;		// linked via attribute 
	{attribute 'TcLinkTo' := 'TIID^Device 2 (EtherCAT)^Term 1 (EK1200)^Term 2 (EL3443)^Total Variant Value In^TxPDO Toggle'}
	MDP5001_341_Total_Variant_Value_In_TxPDO_Toggle			AT%I* : BOOL;		// linked via attribute 
	{attribute 'TcLinkTo' := 'TIID^Device 2 (EtherCAT)^Term 1 (EK1200)^Term 2 (EL3443)^Total Variant Value In^Index 1 REAL'}
	MDP5001_341_Total_Variant_Value_In_Index_1_REAL			AT%I* : UINT;		// linked via attribute 
	{attribute 'TcLinkTo' := 'TIID^Device 2 (EtherCAT)^Term 1 (EK1200)^Term 2 (EL3443)^Total Variant Value In^Value 1 REAL'}
	MDP5001_341_Total_Variant_Value_In_Value_1_REAL			AT%I* : REAL;		// linked via attribute 
	{attribute 'TcLinkTo' := 'TIID^Device 2 (EtherCAT)^Term 1 (EK1200)^Term 2 (EL3443)^Total Variant Value In^Index 2 REAL'}
	MDP5001_341_Total_Variant_Value_In_Index_2_REAL			AT%I* : UINT;		// linked via attribute 
	{attribute 'TcLinkTo' := 'TIID^Device 2 (EtherCAT)^Term 1 (EK1200)^Term 2 (EL3443)^Total Variant Value In^Value 2 REAL'}
	MDP5001_341_Total_Variant_Value_In_Value_2_REAL			AT%I* : REAL;		// linked via attribute 
	{attribute 'TcLinkTo' := 'TIID^Device 2 (EtherCAT)^Term 1 (EK1200)^Term 2 (EL3443)^Total Variant Value In^Index 3 REAL'}
	MDP5001_341_Total_Variant_Value_In_Index_3_REAL			AT%I* : UINT;		// linked via attribute 
	{attribute 'TcLinkTo' := 'TIID^Device 2 (EtherCAT)^Term 1 (EK1200)^Term 2 (EL3443)^Total Variant Value In^Value 3 REAL'}
	MDP5001_341_Total_Variant_Value_In_Value_3_REAL			AT%I* : REAL;		// linked via attribute 
	{attribute 'TcLinkTo' := 'TIID^Device 2 (EtherCAT)^Term 1 (EK1200)^Term 2 (EL3443)^Total Variant Value In^Index 4 ULINT'}
	MDP5001_341_Total_Variant_Value_In_Index_4_ULINT		AT%I* : UINT;		// linked via attribute 
	{attribute 'TcLinkTo' := 'TIID^Device 2 (EtherCAT)^Term 1 (EK1200)^Term 2 (EL3443)^Total Variant Value In^Value 4 ULINT'}
	MDP5001_341_Total_Variant_Value_In_Value_4_ULINT		AT%I* : ULINT;	// linked via attribute 
	{attribute 'TcLinkTo' := 'TIID^Device 2 (EtherCAT)^Term 1 (EK1200)^Term 2 (EL3443)^DPM Data^Data 1'}
	MDP5001_341_DPM_Data_Data_1								AT%I* : UDINT;	// linked via attribute 
	{attribute 'TcLinkTo' := 'TIID^Device 2 (EtherCAT)^Term 1 (EK1200)^Term 2 (EL3443)^DPM Data^Data 2'}
	MDP5001_341_DPM_Data_Data_2								AT%I* : UDINT;	// linked via attribute 
	{attribute 'TcLinkTo' := 'TIID^Device 2 (EtherCAT)^Term 1 (EK1200)^Term 2 (EL3443)^DPM Data^Data 3'}
	MDP5001_341_DPM_Data_Data_3								AT%I* : UDINT;	// linked via attribute 
	{attribute 'TcLinkTo' := 'TIID^Device 2 (EtherCAT)^Term 1 (EK1200)^Term 2 (EL3443)^DPM Data^Data 4'}
	MDP5001_341_DPM_Data_Data_4								AT%I* : UDINT;	// linked via attribute 
	{attribute 'TcLinkTo' := 'TIID^Device 2 (EtherCAT)^Term 1 (EK1200)^Term 2 (EL3443)^DPM Data^Data 5'}
	MDP5001_341_DPM_Data_Data_5								AT%I* : UDINT;	// linked via attribute 
	{attribute 'TcLinkTo' := 'TIID^Device 2 (EtherCAT)^Term 1 (EK1200)^Term 2 (EL3443)^DPM Data^Data 6'}
	MDP5001_341_DPM_Data_Data_6								AT%I* : UDINT;	// linked via attribute 
	{attribute 'TcLinkTo' := 'TIID^Device 2 (EtherCAT)^Term 1 (EK1200)^Term 2 (EL3443)^DPM Data^Data 7'}
	MDP5001_341_DPM_Data_Data_7								AT%I* : UDINT;	// linked via attribute 
	{attribute 'TcLinkTo' := 'TIID^Device 2 (EtherCAT)^Term 1 (EK1200)^Term 2 (EL3443)^DPM Data^Data 8'}
	MDP5001_341_DPM_Data_Data_8								AT%I* : UDINT;	// linked via attribute 
	{attribute 'TcLinkTo' := 'TIID^Device 2 (EtherCAT)^Term 1 (EK1200)^Term 2 (EL3443)^DPM Data^Data 9'}
	MDP5001_341_DPM_Data_Data_9								AT%I* : UDINT;	// linked via attribute 
	{attribute 'TcLinkTo' := 'TIID^Device 2 (EtherCAT)^Term 1 (EK1200)^Term 2 (EL3443)^DPM Data^Data 10'}
	MDP5001_341_DPM_Data_Data_10							AT%I* : UDINT;	// linked via attribute 
	{attribute 'TcLinkTo' := 'TIID^Device 2 (EtherCAT)^Term 1 (EK1200)^Term 2 (EL3443)^DPM Data^Data 11'}
	MDP5001_341_DPM_Data_Data_11							AT%I* : UDINT;	// linked via attribute 
	{attribute 'TcLinkTo' := 'TIID^Device 2 (EtherCAT)^Term 1 (EK1200)^Term 2 (EL3443)^DPM Data^Data 12'}
	MDP5001_341_DPM_Data_Data_12							AT%I* : UDINT;	// linked via attribute 
	{attribute 'TcLinkTo' := 'TIID^Device 2 (EtherCAT)^Term 1 (EK1200)^Term 2 (EL3443)^DPM Data^Data 13'}
	MDP5001_341_DPM_Data_Data_13							AT%I* : UDINT;	// linked via attribute 
	{attribute 'TcLinkTo' := 'TIID^Device 2 (EtherCAT)^Term 1 (EK1200)^Term 2 (EL3443)^DPM Data^Data 14'}
	MDP5001_341_DPM_Data_Data_14							AT%I* : UDINT;	// linked via attribute 
	{attribute 'TcLinkTo' := 'TIID^Device 2 (EtherCAT)^Term 1 (EK1200)^Term 2 (EL3443)^DPM Data^Data 15'}
	MDP5001_341_DPM_Data_Data_15							AT%I* : UDINT;	// linked via attribute 
	{attribute 'TcLinkTo' := 'TIID^Device 2 (EtherCAT)^Term 1 (EK1200)^Term 2 (EL3443)^DPM Data^Data 16'}
	MDP5001_341_DPM_Data_Data_16							AT%I* : UDINT;	// linked via attribute 
	{attribute 'TcLinkTo' := 'TIID^Device 2 (EtherCAT)^Term 1 (EK1200)^Term 2 (EL3443)^DPM Data^Data 17'}
	MDP5001_341_DPM_Data_Data_17							AT%I* : UDINT;	// linked via attribute 
	{attribute 'TcLinkTo' := 'TIID^Device 2 (EtherCAT)^Term 1 (EK1200)^Term 2 (EL3443)^DPM Data^Data 18'}
	MDP5001_341_DPM_Data_Data_18							AT%I* : UDINT;	// linked via attribute 
	{attribute 'TcLinkTo' := 'TIID^Device 2 (EtherCAT)^Term 1 (EK1200)^Term 2 (EL3443)^DPM Data^Data 19'}
	MDP5001_341_DPM_Data_Data_19							AT%I* : UDINT;	// linked via attribute 
	{attribute 'TcLinkTo' := 'TIID^Device 2 (EtherCAT)^Term 1 (EK1200)^Term 2 (EL3443)^DPM Data^Data 20'}
	MDP5001_341_DPM_Data_Data_20							AT%I* : UDINT;	// linked via attribute 
	{attribute 'TcLinkTo' := 'TIID^Device 2 (EtherCAT)^Term 1 (EK1200)^Term 2 (EL3443)^Total Variant Value Out^Index 1 REAL'}
	MDP5001_341_Total_Variant_Value_Out_Index_1_REAL	AT%Q* : UINT;
	{attribute 'TcLinkTo' := 'TIID^Device 2 (EtherCAT)^Term 1 (EK1200)^Term 2 (EL3443)^Total Variant Value Out^Index 2 REAL'}
	MDP5001_341_Total_Variant_Value_Out_Index_2_REAL	AT%Q* : UINT;
	{attribute 'TcLinkTo' := 'TIID^Device 2 (EtherCAT)^Term 1 (EK1200)^Term 2 (EL3443)^Total Variant Value Out^Index 3 REAL'}
	MDP5001_341_Total_Variant_Value_Out_Index_3_REAL	AT%Q* : UINT;
	{attribute 'TcLinkTo' := 'TIID^Device 2 (EtherCAT)^Term 1 (EK1200)^Term 2 (EL3443)^Total Variant Value Out^Index 4 ULINT'}
	MDP5001_341_Total_Variant_Value_Out_Index_4_ULINT	AT%Q* : UINT;
	{attribute 'TcLinkTo' := 'TIID^Device 2 (EtherCAT)^Term 1 (EK1200)^Term 2 (EL3443)^Total Interval^Reset Interval'}
	MDP5001_341_Total_Interval_Reset_Interval			AT%Q* : BOOL;	

	
// IOs for EL3446-1
	{attribute 'TcLinkTo' := 'TIID^Device 2 (EtherCAT)^Term 1 (EK1200)^Term 3 (EL3446)^I1 Channel^Overcurrent'}
	MDP5001_342_I1_Channel_Overcurrent_EM1						AT%I*  : BOOL;
	{attribute 'TcLinkTo' := 'TIID^Device 2 (EtherCAT)^Term 1 (EK1200)^Term 3 (EL3446)^I1 Channel^Inaccurate Current'}
	MDP5001_342_I1_Channel_Inaccurate_Current_EM1				AT%I*  : BOOL;
	{attribute 'TcLinkTo' := 'TIID^Device 2 (EtherCAT)^Term 1 (EK1200)^Term 3 (EL3446)^I1 Channel^Current Guard Warning'}
	MDP5001_342_I1_Channel_Current_Guard_Warning_EM1			AT%I*  : BOOL;
	{attribute 'TcLinkTo' := 'TIID^Device 2 (EtherCAT)^Term 1 (EK1200)^Term 3 (EL3446)^I1 Channel^Current Guard Error'}
	MDP5001_342_I1_Channel_Current_Guard_Error_EM1				AT%I*  : BOOL;
	{attribute 'TcLinkTo' := 'TIID^Device 2 (EtherCAT)^Term 1 (EK1200)^Term 3 (EL3446)^I1 Channel^Apparent Power Guard Warning'}
	MDP5001_342_I1_Channel_Apparent_Power_Guard_Warning_EM1		AT%I*  : BOOL;
	{attribute 'TcLinkTo' := 'TIID^Device 2 (EtherCAT)^Term 1 (EK1200)^Term 3 (EL3446)^I1 Channel^Apparent Power Guard Error'}
	MDP5001_342_I1_Channel_Apparent_Power_Guard_Error_EM1		AT%I*  : BOOL;
	{attribute 'TcLinkTo' := 'TIID^Device 2 (EtherCAT)^Term 1 (EK1200)^Term 3 (EL3446)^I1 Channel^Active Power Guard Warning'}
	MDP5001_342_I1_Channel_Active_Power_Guard_Warning_EM1		AT%I*  : BOOL;
	{attribute 'TcLinkTo' := 'TIID^Device 2 (EtherCAT)^Term 1 (EK1200)^Term 3 (EL3446)^I1 Channel^Active Power Guard Error'}
	MDP5001_342_I1_Channel_Active_Power_Guard_Error_EM1			AT%I*  : BOOL;
	{attribute 'TcLinkTo' := 'TIID^Device 2 (EtherCAT)^Term 1 (EK1200)^Term 3 (EL3446)^I1 Channel^Reactive Power Guard Warning'}
	MDP5001_342_I1_Channel_Reactive_Power_Guard_Warning_EM1		AT%I*  : BOOL;
	{attribute 'TcLinkTo' := 'TIID^Device 2 (EtherCAT)^Term 1 (EK1200)^Term 3 (EL3446)^I1 Channel^Reactive Power Guard Error'}
	MDP5001_342_I1_Channel_Reactive_Power_Guard_Error_EM1		AT%I*  : BOOL;
	{attribute 'TcLinkTo' := 'TIID^Device 2 (EtherCAT)^Term 1 (EK1200)^Term 3 (EL3446)^I1 Channel^DPM Inaccurate'}
	MDP5001_342_I1_Channel_DPM_Inaccurate_EM1					AT%I*  : BOOL;
	{attribute 'TcLinkTo' := 'TIID^Device 2 (EtherCAT)^Term 1 (EK1200)^Term 3 (EL3446)^I1 Channel^DPM Timeout'}
	MDP5001_342_I1_Channel_DPM_Timeout_EM1						AT%I*  : BOOL;
	{attribute 'TcLinkTo' := 'TIID^Device 2 (EtherCAT)^Term 1 (EK1200)^Term 3 (EL3446)^I1 Channel^TxPDO Toggle'}
	MDP5001_342_I1_Channel_TxPDO_Toggle_EM1						AT%I*  : BOOL;
	{attribute 'TcLinkTo' := 'TIID^Device 2 (EtherCAT)^Term 1 (EK1200)^Term 3 (EL3446)^I1 Channel^Current'}
	MDP5001_342_I1_Channel_Current_EM1							AT%I*  : REAL;
	{attribute 'TcLinkTo' := 'TIID^Device 2 (EtherCAT)^Term 1 (EK1200)^Term 3 (EL3446)^I1 Channel^Active Power'}
	MDP5001_342_I1_Channel_Active_Power_EM1						AT%I*  : REAL;
	{attribute 'TcLinkTo' := 'TIID^Device 2 (EtherCAT)^Term 1 (EK1200)^Term 3 (EL3446)^I1 Channel^Apparent Power'}
	MDP5001_342_I1_Channel_Apparent_Power_EM1					AT%I*  : REAL;
	{attribute 'TcLinkTo' := 'TIID^Device 2 (EtherCAT)^Term 1 (EK1200)^Term 3 (EL3446)^I1 Channel^Reactive Power Fundamental'}
	MDP5001_342_I1_Channel_Reactive_Power_Fundamental_EM1		AT%I*  : REAL;
	{attribute 'TcLinkTo' := 'TIID^Device 2 (EtherCAT)^Term 1 (EK1200)^Term 3 (EL3446)^I1 Channel^Active Energy'}
	MDP5001_342_I1_Channel_Active_Energy_EM1					AT%I*  : DINT;
	{attribute 'TcLinkTo' := 'TIID^Device 2 (EtherCAT)^Term 1 (EK1200)^Term 3 (EL3446)^I2 Channel^Overcurrent'}
	MDP5001_342_I2_Channel_Overcurrent_EM1						AT%I*  : BOOL;
	{attribute 'TcLinkTo' := 'TIID^Device 2 (EtherCAT)^Term 1 (EK1200)^Term 3 (EL3446)^I2 Channel^Inaccurate Current'}
	MDP5001_342_I2_Channel_Inaccurate_Current_EM1				AT%I*  : BOOL;
	{attribute 'TcLinkTo' := 'TIID^Device 2 (EtherCAT)^Term 1 (EK1200)^Term 3 (EL3446)^I2 Channel^Current Guard Warning'}
	MDP5001_342_I2_Channel_Current_Guard_Warning_EM1			AT%I*  : BOOL;
	{attribute 'TcLinkTo' := 'TIID^Device 2 (EtherCAT)^Term 1 (EK1200)^Term 3 (EL3446)^I2 Channel^Current Guard Error'}
	MDP5001_342_I2_Channel_Current_Guard_Error_EM1				AT%I*  : BOOL;
	{attribute 'TcLinkTo' := 'TIID^Device 2 (EtherCAT)^Term 1 (EK1200)^Term 3 (EL3446)^I2 Channel^Apparent Power Guard Warning'}
	MDP5001_342_I2_Channel_Apparent_Power_Guard_Warning_EM1		AT%I*  : BOOL;
	{attribute 'TcLinkTo' := 'TIID^Device 2 (EtherCAT)^Term 1 (EK1200)^Term 3 (EL3446)^I2 Channel^Apparent Power Guard Error'}
	MDP5001_342_I2_Channel_Apparent_Power_Guard_Error_EM1		AT%I*  : BOOL;
	{attribute 'TcLinkTo' := 'TIID^Device 2 (EtherCAT)^Term 1 (EK1200)^Term 3 (EL3446)^I2 Channel^Active Power Guard Warning'}
	MDP5001_342_I2_Channel_Active_Power_Guard_Warning_EM1		AT%I*  : BOOL;
	{attribute 'TcLinkTo' := 'TIID^Device 2 (EtherCAT)^Term 1 (EK1200)^Term 3 (EL3446)^I2 Channel^Active Power Guard Error'}
	MDP5001_342_I2_Channel_Active_Power_Guard_Error_EM1			AT%I*  : BOOL;
	{attribute 'TcLinkTo' := 'TIID^Device 2 (EtherCAT)^Term 1 (EK1200)^Term 3 (EL3446)^I2 Channel^Reactive Power Guard Warning'}
	MDP5001_342_I2_Channel_Reactive_Power_Guard_Warning_EM1		AT%I*  : BOOL;
	{attribute 'TcLinkTo' := 'TIID^Device 2 (EtherCAT)^Term 1 (EK1200)^Term 3 (EL3446)^I2 Channel^Reactive Power Guard Error'}
	MDP5001_342_I2_Channel_Reactive_Power_Guard_Error_EM1		AT%I*  : BOOL;
	{attribute 'TcLinkTo' := 'TIID^Device 2 (EtherCAT)^Term 1 (EK1200)^Term 3 (EL3446)^I2 Channel^DPM Inaccurate'}
	MDP5001_342_I2_Channel_DPM_Inaccurate_EM1					AT%I*  : BOOL;
	{attribute 'TcLinkTo' := 'TIID^Device 2 (EtherCAT)^Term 1 (EK1200)^Term 3 (EL3446)^I2 Channel^DPM Timeout'}
	MDP5001_342_I2_Channel_DPM_Timeout_EM1						AT%I*  : BOOL;
	{attribute 'TcLinkTo' := 'TIID^Device 2 (EtherCAT)^Term 1 (EK1200)^Term 3 (EL3446)^I2 Channel^TxPDO Toggle'}
	MDP5001_342_I2_Channel_TxPDO_Toggle_EM1						AT%I*  : BOOL;
	{attribute 'TcLinkTo' := 'TIID^Device 2 (EtherCAT)^Term 1 (EK1200)^Term 3 (EL3446)^I2 Channel^Current'}
	MDP5001_342_I2_Channel_Current_EM1							AT%I*  : REAL;
	{attribute 'TcLinkTo' := 'TIID^Device 2 (EtherCAT)^Term 1 (EK1200)^Term 3 (EL3446)^I2 Channel^Active Power'}
	MDP5001_342_I2_Channel_Active_Power_EM1						AT%I*  : REAL;
	{attribute 'TcLinkTo' := 'TIID^Device 2 (EtherCAT)^Term 1 (EK1200)^Term 3 (EL3446)^I2 Channel^Apparent Power'}
	MDP5001_342_I2_Channel_Apparent_Power_EM1					AT%I*  : REAL;
	{attribute 'TcLinkTo' := 'TIID^Device 2 (EtherCAT)^Term 1 (EK1200)^Term 3 (EL3446)^I2 Channel^Reactive Power Fundamental'}
	MDP5001_342_I2_Channel_Reactive_Power_Fundamental_EM1		AT%I*  : REAL;
	{attribute 'TcLinkTo' := 'TIID^Device 2 (EtherCAT)^Term 1 (EK1200)^Term 3 (EL3446)^I2 Channel^Active Energy'}
	MDP5001_342_I2_Channel_Active_Energy_EM1					AT%I*  : DINT;
	{attribute 'TcLinkTo' := 'TIID^Device 2 (EtherCAT)^Term 1 (EK1200)^Term 3 (EL3446)^I3 Channel^Overcurrent'}
	MDP5001_342_I3_Channel_Overcurrent_EM1						AT%I*  : BOOL;
	{attribute 'TcLinkTo' := 'TIID^Device 2 (EtherCAT)^Term 1 (EK1200)^Term 3 (EL3446)^I3 Channel^Inaccurate Current'}
	MDP5001_342_I3_Channel_Inaccurate_Current_EM1				AT%I*  : BOOL;
	{attribute 'TcLinkTo' := 'TIID^Device 2 (EtherCAT)^Term 1 (EK1200)^Term 3 (EL3446)^I3 Channel^Current Guard Warning'}
	MDP5001_342_I3_Channel_Current_Guard_Warning_EM1			AT%I*  : BOOL;
	{attribute 'TcLinkTo' := 'TIID^Device 2 (EtherCAT)^Term 1 (EK1200)^Term 3 (EL3446)^I3 Channel^Current Guard Error'}
	MDP5001_342_I3_Channel_Current_Guard_Error_EM1				AT%I*  : BOOL;
	{attribute 'TcLinkTo' := 'TIID^Device 2 (EtherCAT)^Term 1 (EK1200)^Term 3 (EL3446)^I3 Channel^Apparent Power Guard Warning'}
	MDP5001_342_I3_Channel_Apparent_Power_Guard_Warning_EM1		AT%I*  : BOOL;
	{attribute 'TcLinkTo' := 'TIID^Device 2 (EtherCAT)^Term 1 (EK1200)^Term 3 (EL3446)^I3 Channel^Apparent Power Guard Error'}
	MDP5001_342_I3_Channel_Apparent_Power_Guard_Error_EM1		AT%I*  : BOOL;
	{attribute 'TcLinkTo' := 'TIID^Device 2 (EtherCAT)^Term 1 (EK1200)^Term 3 (EL3446)^I3 Channel^Active Power Guard Warning'}
	MDP5001_342_I3_Channel_Active_Power_Guard_Warning_EM1		AT%I*  : BOOL;
	{attribute 'TcLinkTo' := 'TIID^Device 2 (EtherCAT)^Term 1 (EK1200)^Term 3 (EL3446)^I3 Channel^Active Power Guard Error'}
	MDP5001_342_I3_Channel_Active_Power_Guard_Error_EM1		AT%I*  : BOOL;
	{attribute 'TcLinkTo' := 'TIID^Device 2 (EtherCAT)^Term 1 (EK1200)^Term 3 (EL3446)^I3 Channel^Reactive Power Guard Warning'}
	MDP5001_342_I3_Channel_Reactive_Power_Guard_Warning_EM1		AT%I*  : BOOL;
	{attribute 'TcLinkTo' := 'TIID^Device 2 (EtherCAT)^Term 1 (EK1200)^Term 3 (EL3446)^I3 Channel^Reactive Power Guard Error'}
	MDP5001_342_I3_Channel_Reactive_Power_Guard_Error_EM1		AT%I*  : BOOL;
	{attribute 'TcLinkTo' := 'TIID^Device 2 (EtherCAT)^Term 1 (EK1200)^Term 3 (EL3446)^I3 Channel^DPM Inaccurate'}
	MDP5001_342_I3_Channel_DPM_Inaccurate_EM1					AT%I*  : BOOL;
	{attribute 'TcLinkTo' := 'TIID^Device 2 (EtherCAT)^Term 1 (EK1200)^Term 3 (EL3446)^I3 Channel^DPM Timeout'}
	MDP5001_342_I3_Channel_DPM_Timeout_EM1						AT%I*  : BOOL;
	{attribute 'TcLinkTo' := 'TIID^Device 2 (EtherCAT)^Term 1 (EK1200)^Term 3 (EL3446)^I3 Channel^TxPDO Toggle'}
	MDP5001_342_I3_Channel_TxPDO_Toggle_EM1						AT%I*  : BOOL;
	{attribute 'TcLinkTo' := 'TIID^Device 2 (EtherCAT)^Term 1 (EK1200)^Term 3 (EL3446)^I3 Channel^Current'}
	MDP5001_342_I3_Channel_Current_EM1							AT%I*  : REAL;
	{attribute 'TcLinkTo' := 'TIID^Device 2 (EtherCAT)^Term 1 (EK1200)^Term 3 (EL3446)^I3 Channel^Active Power'}
	MDP5001_342_I3_Channel_Active_Power_EM1						AT%I*  : REAL;
	{attribute 'TcLinkTo' := 'TIID^Device 2 (EtherCAT)^Term 1 (EK1200)^Term 3 (EL3446)^I3 Channel^Apparent Power'}
	MDP5001_342_I3_Channel_Apparent_Power_EM1					AT%I*  : REAL;
	{attribute 'TcLinkTo' := 'TIID^Device 2 (EtherCAT)^Term 1 (EK1200)^Term 3 (EL3446)^I3 Channel^Reactive Power Fundamental'}
	MDP5001_342_I3_Channel_Reactive_Power_Fundamental_EM1		AT%I*  : REAL;
	{attribute 'TcLinkTo' := 'TIID^Device 2 (EtherCAT)^Term 1 (EK1200)^Term 3 (EL3446)^I3 Channel^Active Energy'}
	MDP5001_342_I3_Channel_Active_Energy_EM1					AT%I*  : DINT;	
	{attribute 'TcLinkTo' := 'TIID^Device 2 (EtherCAT)^Term 1 (EK1200)^Term 3 (EL3446)^I4 Channel^Overcurrent'}
	MDP5001_342_I4_Channel_Overcurrent_EM1						AT%I*  : BOOL;
	{attribute 'TcLinkTo' := 'TIID^Device 2 (EtherCAT)^Term 1 (EK1200)^Term 3 (EL3446)^I4 Channel^Inaccurate Current'}
	MDP5001_342_I4_Channel_Inaccurate_Current_EM1				AT%I*  : BOOL;
	{attribute 'TcLinkTo' := 'TIID^Device 2 (EtherCAT)^Term 1 (EK1200)^Term 3 (EL3446)^I4 Channel^Current Guard Warning'}
	MDP5001_342_I4_Channel_Current_Guard_Warning_EM1			AT%I*  : BOOL;
	{attribute 'TcLinkTo' := 'TIID^Device 2 (EtherCAT)^Term 1 (EK1200)^Term 3 (EL3446)^I4 Channel^Current Guard Error'}
	MDP5001_342_I4_Channel_Current_Guard_Error_EM1				AT%I*  : BOOL;
	{attribute 'TcLinkTo' := 'TIID^Device 2 (EtherCAT)^Term 1 (EK1200)^Term 3 (EL3446)^I4 Channel^Apparent Power Guard Warning'}
	MDP5001_342_I4_Channel_Apparent_Power_Guard_Warning_EM1		AT%I*  : BOOL;
	{attribute 'TcLinkTo' := 'TIID^Device 2 (EtherCAT)^Term 1 (EK1200)^Term 3 (EL3446)^I4 Channel^Apparent Power Guard Error'}
	MDP5001_342_I4_Channel_Apparent_Power_Guard_Error_EM1		AT%I*  : BOOL;
	{attribute 'TcLinkTo' := 'TIID^Device 2 (EtherCAT)^Term 1 (EK1200)^Term 3 (EL3446)^I4 Channel^Active Power Guard Warning'}
	MDP5001_342_I4_Channel_Active_Power_Guard_Warning_EM1		AT%I*  : BOOL;
	{attribute 'TcLinkTo' := 'TIID^Device 2 (EtherCAT)^Term 1 (EK1200)^Term 3 (EL3446)^I4 Channel^Active Power Guard Error'}
	MDP5001_342_I4_Channel_Active_Power_Guard_Error_EM1			AT%I*  : BOOL;
	{attribute 'TcLinkTo' := 'TIID^Device 2 (EtherCAT)^Term 1 (EK1200)^Term 3 (EL3446)^I4 Channel^Reactive Power Guard Warning'}
	MDP5001_342_I4_Channel_Reactive_Power_Guard_Warning_EM1		AT%I*  : BOOL;
	{attribute 'TcLinkTo' := 'TIID^Device 2 (EtherCAT)^Term 1 (EK1200)^Term 3 (EL3446)^I4 Channel^Reactive Power Guard Error'}
	MDP5001_342_I4_Channel_Reactive_Power_Guard_Error_EM1		AT%I*  : BOOL;
	{attribute 'TcLinkTo' := 'TIID^Device 2 (EtherCAT)^Term 1 (EK1200)^Term 3 (EL3446)^I4 Channel^DPM Inaccurate'}
	MDP5001_342_I4_Channel_DPM_Inaccurate_EM1					AT%I*  : BOOL;
	{attribute 'TcLinkTo' := 'TIID^Device 2 (EtherCAT)^Term 1 (EK1200)^Term 3 (EL3446)^I4 Channel^DPM Timeout'}
	MDP5001_342_I4_Channel_DPM_Timeout_EM1						AT%I*  : BOOL;
	{attribute 'TcLinkTo' := 'TIID^Device 2 (EtherCAT)^Term 1 (EK1200)^Term 3 (EL3446)^I4 Channel^TxPDO Toggle'}
	MDP5001_342_I4_Channel_TxPDO_Toggle_EM1						AT%I*  : BOOL;
	{attribute 'TcLinkTo' := 'TIID^Device 2 (EtherCAT)^Term 1 (EK1200)^Term 3 (EL3446)^I4 Channel^Current'}
	MDP5001_342_I4_Channel_Current_EM1							AT%I*  : REAL;
	{attribute 'TcLinkTo' := 'TIID^Device 2 (EtherCAT)^Term 1 (EK1200)^Term 3 (EL3446)^I4 Channel^Active Power'}
	MDP5001_342_I4_Channel_Active_Power_EM1						AT%I*  : REAL;
	{attribute 'TcLinkTo' := 'TIID^Device 2 (EtherCAT)^Term 1 (EK1200)^Term 3 (EL3446)^I4 Channel^Apparent Power'}
	MDP5001_342_I4_Channel_Apparent_Power_EM1					AT%I*  : REAL;
	{attribute 'TcLinkTo' := 'TIID^Device 2 (EtherCAT)^Term 1 (EK1200)^Term 3 (EL3446)^I4 Channel^Reactive Power Fundamental'}
	MDP5001_342_I4_Channel_Reactive_Power_Fundamental_EM1		AT%I*  : REAL;
	{attribute 'TcLinkTo' := 'TIID^Device 2 (EtherCAT)^Term 1 (EK1200)^Term 3 (EL3446)^I4 Channel^Active Energy'}
	MDP5001_342_I4_Channel_Active_Energy_EM1					AT%I*  : DINT;
	{attribute 'TcLinkTo' := 'TIID^Device 2 (EtherCAT)^Term 1 (EK1200)^Term 3 (EL3446)^I5 Channel^Overcurrent'}
	MDP5001_342_I5_Channel_Overcurrent_EM1						AT%I*  : BOOL;
	{attribute 'TcLinkTo' := 'TIID^Device 2 (EtherCAT)^Term 1 (EK1200)^Term 3 (EL3446)^I5 Channel^Inaccurate Current'}
	MDP5001_342_I5_Channel_Inaccurate_Current_EM1				AT%I*  : BOOL;
	{attribute 'TcLinkTo' := 'TIID^Device 2 (EtherCAT)^Term 1 (EK1200)^Term 3 (EL3446)^I5 Channel^Current Guard Warning'}
	MDP5001_342_I5_Channel_Current_Guard_Warning_EM1			AT%I*  : BOOL;
	{attribute 'TcLinkTo' := 'TIID^Device 2 (EtherCAT)^Term 1 (EK1200)^Term 3 (EL3446)^I5 Channel^Current Guard Error'}
	MDP5001_342_I5_Channel_Current_Guard_Error_EM1				AT%I*  : BOOL;
	{attribute 'TcLinkTo' := 'TIID^Device 2 (EtherCAT)^Term 1 (EK1200)^Term 3 (EL3446)^I5 Channel^Apparent Power Guard Warning'}
	MDP5001_342_I5_Channel_Apparent_Power_Guard_Warning_EM1		AT%I*  : BOOL;
	{attribute 'TcLinkTo' := 'TIID^Device 2 (EtherCAT)^Term 1 (EK1200)^Term 3 (EL3446)^I5 Channel^Apparent Power Guard Error'}
	MDP5001_342_I5_Channel_Apparent_Power_Guard_Error_EM1		AT%I*  : BOOL;
	{attribute 'TcLinkTo' := 'TIID^Device 2 (EtherCAT)^Term 1 (EK1200)^Term 3 (EL3446)^I5 Channel^Active Power Guard Warning'}
	MDP5001_342_I5_Channel_Active_Power_Guard_Warning_EM1		AT%I*  : BOOL;
	{attribute 'TcLinkTo' := 'TIID^Device 2 (EtherCAT)^Term 1 (EK1200)^Term 3 (EL3446)^I5 Channel^Active Power Guard Error'}
	MDP5001_342_I5_Channel_Active_Power_Guard_Error_EM1			AT%I*  : BOOL;
	{attribute 'TcLinkTo' := 'TIID^Device 2 (EtherCAT)^Term 1 (EK1200)^Term 3 (EL3446)^I5 Channel^Reactive Power Guard Warning'}
	MDP5001_342_I5_Channel_Reactive_Power_Guard_Warning_EM1		AT%I*  : BOOL;
	{attribute 'TcLinkTo' := 'TIID^Device 2 (EtherCAT)^Term 1 (EK1200)^Term 3 (EL3446)^I5 Channel^Reactive Power Guard Error'}
	MDP5001_342_I5_Channel_Reactive_Power_Guard_Error_EM1		AT%I*  : BOOL;
	{attribute 'TcLinkTo' := 'TIID^Device 2 (EtherCAT)^Term 1 (EK1200)^Term 3 (EL3446)^I5 Channel^DPM Inaccurate'}
	MDP5001_342_I5_Channel_DPM_Inaccurate_EM1					AT%I*  : BOOL;
	{attribute 'TcLinkTo' := 'TIID^Device 2 (EtherCAT)^Term 1 (EK1200)^Term 3 (EL3446)^I5 Channel^DPM Timeout'}
	MDP5001_342_I5_Channel_DPM_Timeout_EM1						AT%I*  : BOOL;
	{attribute 'TcLinkTo' := 'TIID^Device 2 (EtherCAT)^Term 1 (EK1200)^Term 3 (EL3446)^I5 Channel^TxPDO Toggle'}
	MDP5001_342_I5_Channel_TxPDO_Toggle_EM1						AT%I*  : BOOL;
	{attribute 'TcLinkTo' := 'TIID^Device 2 (EtherCAT)^Term 1 (EK1200)^Term 3 (EL3446)^I5 Channel^Current'}
	MDP5001_342_I5_Channel_Current_EM1							AT%I*  : REAL;
	{attribute 'TcLinkTo' := 'TIID^Device 2 (EtherCAT)^Term 1 (EK1200)^Term 3 (EL3446)^I5 Channel^Active Power'}
	MDP5001_342_I5_Channel_Active_Power_EM1						AT%I*  : REAL;
	{attribute 'TcLinkTo' := 'TIID^Device 2 (EtherCAT)^Term 1 (EK1200)^Term 3 (EL3446)^I5 Channel^Apparent Power'}
	MDP5001_342_I5_Channel_Apparent_Power_EM1					AT%I*  : REAL;
	{attribute 'TcLinkTo' := 'TIID^Device 2 (EtherCAT)^Term 1 (EK1200)^Term 3 (EL3446)^I5 Channel^Reactive Power Fundamental'}
	MDP5001_342_I5_Channel_Reactive_Power_Fundamental_EM1		AT%I*  : REAL;
	{attribute 'TcLinkTo' := 'TIID^Device 2 (EtherCAT)^Term 1 (EK1200)^Term 3 (EL3446)^I5 Channel^Active Energy'}
	MDP5001_342_I5_Channel_Active_Energy_EM1					AT%I*  : DINT;
	{attribute 'TcLinkTo' := 'TIID^Device 2 (EtherCAT)^Term 1 (EK1200)^Term 3 (EL3446)^I6 Channel^Overcurrent'}
	MDP5001_342_I6_Channel_Overcurrent_EM1						AT%I*  : BOOL;
	{attribute 'TcLinkTo' := 'TIID^Device 2 (EtherCAT)^Term 1 (EK1200)^Term 3 (EL3446)^I6 Channel^Inaccurate Current'}
	MDP5001_342_I6_Channel_Inaccurate_Current_EM1				AT%I*  : BOOL;
	{attribute 'TcLinkTo' := 'TIID^Device 2 (EtherCAT)^Term 1 (EK1200)^Term 3 (EL3446)^I6 Channel^Current Guard Warning'}
	MDP5001_342_I6_Channel_Current_Guard_Warning_EM1			AT%I*  : BOOL;
	{attribute 'TcLinkTo' := 'TIID^Device 2 (EtherCAT)^Term 1 (EK1200)^Term 3 (EL3446)^I6 Channel^Current Guard Error'}
	MDP5001_342_I6_Channel_Current_Guard_Error_EM1				AT%I*  : BOOL;
	{attribute 'TcLinkTo' := 'TIID^Device 2 (EtherCAT)^Term 1 (EK1200)^Term 3 (EL3446)^I6 Channel^Apparent Power Guard Warning'}
	MDP5001_342_I6_Channel_Apparent_Power_Guard_Warning_EM1		AT%I*  : BOOL;
	{attribute 'TcLinkTo' := 'TIID^Device 2 (EtherCAT)^Term 1 (EK1200)^Term 3 (EL3446)^I6 Channel^Apparent Power Guard Error'}
	MDP5001_342_I6_Channel_Apparent_Power_Guard_Error_EM1		AT%I*  : BOOL;
	{attribute 'TcLinkTo' := 'TIID^Device 2 (EtherCAT)^Term 1 (EK1200)^Term 3 (EL3446)^I6 Channel^Active Power Guard Warning'}
	MDP5001_342_I6_Channel_Active_Power_Guard_Warning_EM1		AT%I*  : BOOL;
	{attribute 'TcLinkTo' := 'TIID^Device 2 (EtherCAT)^Term 1 (EK1200)^Term 3 (EL3446)^I6 Channel^Active Power Guard Error'}
	MDP5001_342_I6_Channel_Active_Power_Guard_Error_EM1			AT%I*  : BOOL;
	{attribute 'TcLinkTo' := 'TIID^Device 2 (EtherCAT)^Term 1 (EK1200)^Term 3 (EL3446)^I6 Channel^Reactive Power Guard Warning'}
	MDP5001_342_I6_Channel_Reactive_Power_Guard_Warning_EM1		AT%I*  : BOOL;
	{attribute 'TcLinkTo' := 'TIID^Device 2 (EtherCAT)^Term 1 (EK1200)^Term 3 (EL3446)^I6 Channel^Reactive Power Guard Error'}
	MDP5001_342_I6_Channel_Reactive_Power_Guard_Error_EM1		AT%I*  : BOOL;
	{attribute 'TcLinkTo' := 'TIID^Device 2 (EtherCAT)^Term 1 (EK1200)^Term 3 (EL3446)^I6 Channel^DPM Inaccurate'}
	MDP5001_342_I6_Channel_DPM_Inaccurate_EM1					AT%I*  : BOOL;
	{attribute 'TcLinkTo' := 'TIID^Device 2 (EtherCAT)^Term 1 (EK1200)^Term 3 (EL3446)^I6 Channel^DPM Timeout'}
	MDP5001_342_I6_Channel_DPM_Timeout_EM1						AT%I*  : BOOL;
	{attribute 'TcLinkTo' := 'TIID^Device 2 (EtherCAT)^Term 1 (EK1200)^Term 3 (EL3446)^I6 Channel^TxPDO Toggle'}
	MDP5001_342_I6_Channel_TxPDO_Toggle_EM1						AT%I*  : BOOL;
	{attribute 'TcLinkTo' := 'TIID^Device 2 (EtherCAT)^Term 1 (EK1200)^Term 3 (EL3446)^I6 Channel^Current'}
	MDP5001_342_I6_Channel_Current_EM1							AT%I*  : REAL;
	{attribute 'TcLinkTo' := 'TIID^Device 2 (EtherCAT)^Term 1 (EK1200)^Term 3 (EL3446)^I6 Channel^Active Power'}
	MDP5001_342_I6_Channel_Active_Power_EM1						AT%I*  : REAL;
	{attribute 'TcLinkTo' := 'TIID^Device 2 (EtherCAT)^Term 1 (EK1200)^Term 3 (EL3446)^I6 Channel^Apparent Power'}
	MDP5001_342_I6_Channel_Apparent_Power_EM1					AT%I*  : REAL;
	{attribute 'TcLinkTo' := 'TIID^Device 2 (EtherCAT)^Term 1 (EK1200)^Term 3 (EL3446)^I6 Channel^Reactive Power Fundamental'}
	MDP5001_342_I6_Channel_Reactive_Power_Fundamental_EM1		AT%I*  : REAL;
	{attribute 'TcLinkTo' := 'TIID^Device 2 (EtherCAT)^Term 1 (EK1200)^Term 3 (EL3446)^I6 Channel^Active Energy'}
	MDP5001_342_I6_Channel_Active_Energy_EM1					AT%I*  : DINT;	
	
	{attribute 'TcLinkTo' := 'TIID^Device 2 (EtherCAT)^Term 1 (EK1200)^Term 3 (EL3446)^DPM Variant Value In^TxPDO Toggle'}
	MDP5001_342_DPM_Variant_Value_In_TxPDO_Toggle_EM1			AT%I*  : BOOL;
	{attribute 'TcLinkTo' := 'TIID^Device 2 (EtherCAT)^Term 1 (EK1200)^Term 3 (EL3446)^DPM Variant Value In^Index 1 REAL'}
	MDP5001_342_DPM_Variant_Value_In_Index_1_REAL_EM1			AT%I*  : UINT;
	{attribute 'TcLinkTo' := 'TIID^Device 2 (EtherCAT)^Term 1 (EK1200)^Term 3 (EL3446)^DPM Variant Value In^Value 1 REAL'}
	MDP5001_342_DPM_Variant_Value_In_Value_1_REAL_EM1			AT%I*  : REAL;
	{attribute 'TcLinkTo' := 'TIID^Device 2 (EtherCAT)^Term 1 (EK1200)^Term 3 (EL3446)^DPM Variant Value In^Index 2 REAL'}
	MDP5001_342_DPM_Variant_Value_In_Index_2_REAL_EM1			AT%I*  : UINT;
	{attribute 'TcLinkTo' := 'TIID^Device 2 (EtherCAT)^Term 1 (EK1200)^Term 3 (EL3446)^DPM Variant Value In^Value 2 REAL'}
	MDP5001_342_DPM_Variant_Value_In_Value_2_REAL_EM1			AT%I*  : REAL;
	{attribute 'TcLinkTo' := 'TIID^Device 2 (EtherCAT)^Term 1 (EK1200)^Term 3 (EL3446)^DPM Variant Value In^Index 3 REAL'}
	MDP5001_342_DPM_Variant_Value_In_Index_3_REAL_EM1			AT%I*  : UINT;
	{attribute 'TcLinkTo' := 'TIID^Device 2 (EtherCAT)^Term 1 (EK1200)^Term 3 (EL3446)^DPM Variant Value In^Value 3 REAL'}
	MDP5001_342_DPM_Variant_Value_In_Value_3_REAL_EM1			AT%I*  : REAL;
	{attribute 'TcLinkTo' := 'TIID^Device 2 (EtherCAT)^Term 1 (EK1200)^Term 3 (EL3446)^DPM Variant Value In^Index 4 ULINT'}
	MDP5001_342_DPM_Variant_Value_In_Index_4_ULINT_EM1			AT%I*  : UINT;
	{attribute 'TcLinkTo' := 'TIID^Device 2 (EtherCAT)^Term 1 (EK1200)^Term 3 (EL3446)^DPM Variant Value In^Value 4 ULINT'}
	MDP5001_342_DPM_Variant_Value_In_Value_4_ULINT_EM1			AT%I*  : ULINT;

	{attribute 'TcLinkTo' := 'TIID^Device 2 (EtherCAT)^Term 1 (EK1200)^Term 3 (EL3446)^DPM Variant Value Out^Index 1 REAL'}
	MDP5001_342_DPM_Variant_Value_Out_Index_1_REAL_EM1	AT%Q* : UINT;
	{attribute 'TcLinkTo' := 'TIID^Device 2 (EtherCAT)^Term 1 (EK1200)^Term 3 (EL3446)^DPM Variant Value Out^Index 2 REAL'}
	MDP5001_342_DPM_Variant_Value_Out_Index_2_REAL_EM1	AT%Q* : UINT;
	{attribute 'TcLinkTo' := 'TIID^Device 2 (EtherCAT)^Term 1 (EK1200)^Term 3 (EL3446)^DPM Variant Value Out^Index 3 REAL'}
	MDP5001_342_DPM_Variant_Value_Out_Index_3_REAL_EM1	AT%Q* : UINT;
	{attribute 'TcLinkTo' := 'TIID^Device 2 (EtherCAT)^Term 1 (EK1200)^Term 3 (EL3446)^DPM Variant Value Out^Index 4 ULINT'}
	MDP5001_342_DPM_Variant_Value_Out_Index_4_ULINT_EM1	AT%Q* : UINT;
	{attribute 'TcLinkTo' := 'TIID^Device 2 (EtherCAT)^Term 1 (EK1200)^Term 3 (EL3446)^DPM Data^Data 1'}
	MDP5001_342_DPM_Data_Data_1_EM1						AT%Q* : UDINT;
	{attribute 'TcLinkTo' := 'TIID^Device 2 (EtherCAT)^Term 1 (EK1200)^Term 3 (EL3446)^DPM Data^Data 2'}
	MDP5001_342_DPM_Data_Data_2_EM1						AT%Q* : UDINT;
	{attribute 'TcLinkTo' := 'TIID^Device 2 (EtherCAT)^Term 1 (EK1200)^Term 3 (EL3446)^DPM Data^Data 3'}
	MDP5001_342_DPM_Data_Data_3_EM1						AT%Q* : UDINT;
	{attribute 'TcLinkTo' := 'TIID^Device 2 (EtherCAT)^Term 1 (EK1200)^Term 3 (EL3446)^DPM Data^Data 4'}
	MDP5001_342_DPM_Data_Data_4_EM1						AT%Q* : UDINT;
	{attribute 'TcLinkTo' := 'TIID^Device 2 (EtherCAT)^Term 1 (EK1200)^Term 3 (EL3446)^DPM Data^Data 5'}
	MDP5001_342_DPM_Data_Data_5_EM1						AT%Q* : UDINT;
	{attribute 'TcLinkTo' := 'TIID^Device 2 (EtherCAT)^Term 1 (EK1200)^Term 3 (EL3446)^DPM Data^Data 6'}
	MDP5001_342_DPM_Data_Data_6_EM1						AT%Q* : UDINT;
	{attribute 'TcLinkTo' := 'TIID^Device 2 (EtherCAT)^Term 1 (EK1200)^Term 3 (EL3446)^DPM Data^Data 7'}
	MDP5001_342_DPM_Data_Data_7_EM1						AT%Q* : UDINT;
	{attribute 'TcLinkTo' := 'TIID^Device 2 (EtherCAT)^Term 1 (EK1200)^Term 3 (EL3446)^DPM Data^Data 8'}
	MDP5001_342_DPM_Data_Data_8_EM1						AT%Q* : UDINT;
	{attribute 'TcLinkTo' := 'TIID^Device 2 (EtherCAT)^Term 1 (EK1200)^Term 3 (EL3446)^DPM Data^Data 9'}
	MDP5001_342_DPM_Data_Data_9_EM1						AT%Q* : UDINT;
	{attribute 'TcLinkTo' := 'TIID^Device 2 (EtherCAT)^Term 1 (EK1200)^Term 3 (EL3446)^DPM Data^Data 10'}
	MDP5001_342_DPM_Data_Data_10_EM1					AT%Q* : UDINT;
	{attribute 'TcLinkTo' := 'TIID^Device 2 (EtherCAT)^Term 1 (EK1200)^Term 3 (EL3446)^DPM Data^Data 11'}
	MDP5001_342_DPM_Data_Data_11_EM1					AT%Q* : UDINT;
	{attribute 'TcLinkTo' := 'TIID^Device 2 (EtherCAT)^Term 1 (EK1200)^Term 3 (EL3446)^DPM Data^Data 12'}
	MDP5001_342_DPM_Data_Data_12_EM1					AT%Q* : UDINT;
	{attribute 'TcLinkTo' := 'TIID^Device 2 (EtherCAT)^Term 1 (EK1200)^Term 3 (EL3446)^DPM Data^Data 13'}
	MDP5001_342_DPM_Data_Data_13_EM1					AT%Q* : UDINT;
	{attribute 'TcLinkTo' := 'TIID^Device 2 (EtherCAT)^Term 1 (EK1200)^Term 3 (EL3446)^DPM Data^Data 14'}
	MDP5001_342_DPM_Data_Data_14_EM1					AT%Q* : UDINT;
	{attribute 'TcLinkTo' := 'TIID^Device 2 (EtherCAT)^Term 1 (EK1200)^Term 3 (EL3446)^DPM Data^Data 15'}
	MDP5001_342_DPM_Data_Data_15_EM1					AT%Q* : UDINT;
	{attribute 'TcLinkTo' := 'TIID^Device 2 (EtherCAT)^Term 1 (EK1200)^Term 3 (EL3446)^DPM Data^Data 16'}
	MDP5001_342_DPM_Data_Data_16_EM1					AT%Q* : UDINT;
	{attribute 'TcLinkTo' := 'TIID^Device 2 (EtherCAT)^Term 1 (EK1200)^Term 3 (EL3446)^DPM Data^Data 17'}
	MDP5001_342_DPM_Data_Data_17_EM1					AT%Q* : UDINT;
	{attribute 'TcLinkTo' := 'TIID^Device 2 (EtherCAT)^Term 1 (EK1200)^Term 3 (EL3446)^DPM Data^Data 18'}
	MDP5001_342_DPM_Data_Data_18_EM1					AT%Q* : UDINT;
	{attribute 'TcLinkTo' := 'TIID^Device 2 (EtherCAT)^Term 1 (EK1200)^Term 3 (EL3446)^DPM Data^Data 19'}
	MDP5001_342_DPM_Data_Data_19_EM1					AT%Q* : UDINT;
	{attribute 'TcLinkTo' := 'TIID^Device 2 (EtherCAT)^Term 1 (EK1200)^Term 3 (EL3446)^DPM Data^Data 20'}
	MDP5001_342_DPM_Data_Data_20_EM1					AT%Q* : UDINT;

	
// IOs for EL3446-2
	{attribute 'TcLinkTo' := 'TIID^Device 2 (EtherCAT)^Term 1 (EK1200)^Term 4 (EL3446)^I1 Channel^Overcurrent'}
	MDP5001_342_I1_Channel_Overcurrent_EM2						AT%I*  : BOOL;
	{attribute 'TcLinkTo' := 'TIID^Device 2 (EtherCAT)^Term 1 (EK1200)^Term 4 (EL3446)^I1 Channel^Inaccurate Current'}
	MDP5001_342_I1_Channel_Inaccurate_Current_EM2				AT%I*  : BOOL;
	{attribute 'TcLinkTo' := 'TIID^Device 2 (EtherCAT)^Term 1 (EK1200)^Term 4 (EL3446)^I1 Channel^Current Guard Warning'}
	MDP5001_342_I1_Channel_Current_Guard_Warning_EM2			AT%I*  : BOOL;
	{attribute 'TcLinkTo' := 'TIID^Device 2 (EtherCAT)^Term 1 (EK1200)^Term 4 (EL3446)^I1 Channel^Current Guard Error'}
	MDP5001_342_I1_Channel_Current_Guard_Error_EM2				AT%I*  : BOOL;
	{attribute 'TcLinkTo' := 'TIID^Device 2 (EtherCAT)^Term 1 (EK1200)^Term 4 (EL3446)^I1 Channel^Apparent Power Guard Warning'}
	MDP5001_342_I1_Channel_Apparent_Power_Guard_Warning_EM2		AT%I*  : BOOL;
	{attribute 'TcLinkTo' := 'TIID^Device 2 (EtherCAT)^Term 1 (EK1200)^Term 4 (EL3446)^I1 Channel^Apparent Power Guard Error'}
	MDP5001_342_I1_Channel_Apparent_Power_Guard_Error_EM2		AT%I*  : BOOL;
	{attribute 'TcLinkTo' := 'TIID^Device 2 (EtherCAT)^Term 1 (EK1200)^Term 4 (EL3446)^I1 Channel^Active Power Guard Warning'}
	MDP5001_342_I1_Channel_Active_Power_Guard_Warning_EM2		AT%I*  : BOOL;
	{attribute 'TcLinkTo' := 'TIID^Device 2 (EtherCAT)^Term 1 (EK1200)^Term 4 (EL3446)^I1 Channel^Active Power Guard Error'}
	MDP5001_342_I1_Channel_Active_Power_Guard_Error_EM2			AT%I*  : BOOL;
	{attribute 'TcLinkTo' := 'TIID^Device 2 (EtherCAT)^Term 1 (EK1200)^Term 4 (EL3446)^I1 Channel^Reactive Power Guard Warning'}
	MDP5001_342_I1_Channel_Reactive_Power_Guard_Warning_EM2		AT%I*  : BOOL;
	{attribute 'TcLinkTo' := 'TIID^Device 2 (EtherCAT)^Term 1 (EK1200)^Term 4 (EL3446)^I1 Channel^Reactive Power Guard Error'}
	MDP5001_342_I1_Channel_Reactive_Power_Guard_Error_EM2		AT%I*  : BOOL;
	{attribute 'TcLinkTo' := 'TIID^Device 2 (EtherCAT)^Term 1 (EK1200)^Term 4 (EL3446)^I1 Channel^DPM Inaccurate'}
	MDP5001_342_I1_Channel_DPM_Inaccurate_EM2					AT%I*  : BOOL;
	{attribute 'TcLinkTo' := 'TIID^Device 2 (EtherCAT)^Term 1 (EK1200)^Term 4 (EL3446)^I1 Channel^DPM Timeout'}
	MDP5001_342_I1_Channel_DPM_Timeout_EM2						AT%I*  : BOOL;
	{attribute 'TcLinkTo' := 'TIID^Device 2 (EtherCAT)^Term 1 (EK1200)^Term 4 (EL3446)^I1 Channel^TxPDO Toggle'}
	MDP5001_342_I1_Channel_TxPDO_Toggle_EM2						AT%I*  : BOOL;
	{attribute 'TcLinkTo' := 'TIID^Device 2 (EtherCAT)^Term 1 (EK1200)^Term 4 (EL3446)^I1 Channel^Current'}
	MDP5001_342_I1_Channel_Current_EM2							AT%I*  : REAL;
	{attribute 'TcLinkTo' := 'TIID^Device 2 (EtherCAT)^Term 1 (EK1200)^Term 4 (EL3446)^I1 Channel^Active Power'}
	MDP5001_342_I1_Channel_Active_Power_EM2						AT%I*  : REAL;
	{attribute 'TcLinkTo' := 'TIID^Device 2 (EtherCAT)^Term 1 (EK1200)^Term 4 (EL3446)^I1 Channel^Apparent Power'}
	MDP5001_342_I1_Channel_Apparent_Power_EM2					AT%I*  : REAL;
	{attribute 'TcLinkTo' := 'TIID^Device 2 (EtherCAT)^Term 1 (EK1200)^Term 4 (EL3446)^I1 Channel^Reactive Power Fundamental'}
	MDP5001_342_I1_Channel_Reactive_Power_Fundamental_EM2		AT%I*  : REAL;
	{attribute 'TcLinkTo' := 'TIID^Device 2 (EtherCAT)^Term 1 (EK1200)^Term 4 (EL3446)^I1 Channel^Active Energy'}
	MDP5001_342_I1_Channel_Active_Energy_EM2					AT%I*  : DINT;
	{attribute 'TcLinkTo' := 'TIID^Device 2 (EtherCAT)^Term 1 (EK1200)^Term 4 (EL3446)^I2 Channel^Overcurrent'}
	MDP5001_342_I2_Channel_Overcurrent_EM2						AT%I*  : BOOL;
	{attribute 'TcLinkTo' := 'TIID^Device 2 (EtherCAT)^Term 1 (EK1200)^Term 4 (EL3446)^I2 Channel^Inaccurate Current'}
	MDP5001_342_I2_Channel_Inaccurate_Current_EM2				AT%I*  : BOOL;
	{attribute 'TcLinkTo' := 'TIID^Device 2 (EtherCAT)^Term 1 (EK1200)^Term 4 (EL3446)^I2 Channel^Current Guard Warning'}
	MDP5001_342_I2_Channel_Current_Guard_Warning_EM2			AT%I*  : BOOL;
	{attribute 'TcLinkTo' := 'TIID^Device 2 (EtherCAT)^Term 1 (EK1200)^Term 4 (EL3446)^I2 Channel^Current Guard Error'}
	MDP5001_342_I2_Channel_Current_Guard_Error_EM2				AT%I*  : BOOL;
	{attribute 'TcLinkTo' := 'TIID^Device 2 (EtherCAT)^Term 1 (EK1200)^Term 4 (EL3446)^I2 Channel^Apparent Power Guard Warning'}
	MDP5001_342_I2_Channel_Apparent_Power_Guard_Warning_EM2		AT%I*  : BOOL;
	{attribute 'TcLinkTo' := 'TIID^Device 2 (EtherCAT)^Term 1 (EK1200)^Term 4 (EL3446)^I2 Channel^Apparent Power Guard Error'}
	MDP5001_342_I2_Channel_Apparent_Power_Guard_Error_EM2		AT%I*  : BOOL;
	{attribute 'TcLinkTo' := 'TIID^Device 2 (EtherCAT)^Term 1 (EK1200)^Term 4 (EL3446)^I2 Channel^Active Power Guard Warning'}
	MDP5001_342_I2_Channel_Active_Power_Guard_Warning_EM2		AT%I*  : BOOL;
	{attribute 'TcLinkTo' := 'TIID^Device 2 (EtherCAT)^Term 1 (EK1200)^Term 4 (EL3446)^I2 Channel^Active Power Guard Error'}
	MDP5001_342_I2_Channel_Active_Power_Guard_Error_EM2			AT%I*  : BOOL;
	{attribute 'TcLinkTo' := 'TIID^Device 2 (EtherCAT)^Term 1 (EK1200)^Term 4 (EL3446)^I2 Channel^Reactive Power Guard Warning'}
	MDP5001_342_I2_Channel_Reactive_Power_Guard_Warning_EM2		AT%I*  : BOOL;
	{attribute 'TcLinkTo' := 'TIID^Device 2 (EtherCAT)^Term 1 (EK1200)^Term 4 (EL3446)^I2 Channel^Reactive Power Guard Error'}
	MDP5001_342_I2_Channel_Reactive_Power_Guard_Error_EM2		AT%I*  : BOOL;
	{attribute 'TcLinkTo' := 'TIID^Device 2 (EtherCAT)^Term 1 (EK1200)^Term 4 (EL3446)^I2 Channel^DPM Inaccurate'}
	MDP5001_342_I2_Channel_DPM_Inaccurate_EM2					AT%I*  : BOOL;
	{attribute 'TcLinkTo' := 'TIID^Device 2 (EtherCAT)^Term 1 (EK1200)^Term 4 (EL3446)^I2 Channel^DPM Timeout'}
	MDP5001_342_I2_Channel_DPM_Timeout_EM2						AT%I*  : BOOL;
	{attribute 'TcLinkTo' := 'TIID^Device 2 (EtherCAT)^Term 1 (EK1200)^Term 4 (EL3446)^I2 Channel^TxPDO Toggle'}
	MDP5001_342_I2_Channel_TxPDO_Toggle_EM2						AT%I*  : BOOL;
	{attribute 'TcLinkTo' := 'TIID^Device 2 (EtherCAT)^Term 1 (EK1200)^Term 4 (EL3446)^I2 Channel^Current'}
	MDP5001_342_I2_Channel_Current_EM2							AT%I*  : REAL;
	{attribute 'TcLinkTo' := 'TIID^Device 2 (EtherCAT)^Term 1 (EK1200)^Term 4 (EL3446)^I2 Channel^Active Power'}
	MDP5001_342_I2_Channel_Active_Power_EM2						AT%I*  : REAL;
	{attribute 'TcLinkTo' := 'TIID^Device 2 (EtherCAT)^Term 1 (EK1200)^Term 4 (EL3446)^I2 Channel^Apparent Power'}
	MDP5001_342_I2_Channel_Apparent_Power_EM2					AT%I*  : REAL;
	{attribute 'TcLinkTo' := 'TIID^Device 2 (EtherCAT)^Term 1 (EK1200)^Term 4 (EL3446)^I2 Channel^Reactive Power Fundamental'}
	MDP5001_342_I2_Channel_Reactive_Power_Fundamental_EM2		AT%I*  : REAL;
	{attribute 'TcLinkTo' := 'TIID^Device 2 (EtherCAT)^Term 1 (EK1200)^Term 4 (EL3446)^I2 Channel^Active Energy'}
	MDP5001_342_I2_Channel_Active_Energy_EM2					AT%I*  : DINT;
	{attribute 'TcLinkTo' := 'TIID^Device 2 (EtherCAT)^Term 1 (EK1200)^Term 4 (EL3446)^I3 Channel^Overcurrent'}
	MDP5001_342_I3_Channel_Overcurrent_EM2						AT%I*  : BOOL;
	{attribute 'TcLinkTo' := 'TIID^Device 2 (EtherCAT)^Term 1 (EK1200)^Term 4 (EL3446)^I3 Channel^Inaccurate Current'}
	MDP5001_342_I3_Channel_Inaccurate_Current_EM2				AT%I*  : BOOL;
	{attribute 'TcLinkTo' := 'TIID^Device 2 (EtherCAT)^Term 1 (EK1200)^Term 4 (EL3446)^I3 Channel^Current Guard Warning'}
	MDP5001_342_I3_Channel_Current_Guard_Warning_EM2			AT%I*  : BOOL;
	{attribute 'TcLinkTo' := 'TIID^Device 2 (EtherCAT)^Term 1 (EK1200)^Term 4 (EL3446)^I3 Channel^Current Guard Error'}
	MDP5001_342_I3_Channel_Current_Guard_Error_EM2				AT%I*  : BOOL;
	{attribute 'TcLinkTo' := 'TIID^Device 2 (EtherCAT)^Term 1 (EK1200)^Term 4 (EL3446)^I3 Channel^Apparent Power Guard Warning'}
	MDP5001_342_I3_Channel_Apparent_Power_Guard_Warning_EM2		AT%I*  : BOOL;
	{attribute 'TcLinkTo' := 'TIID^Device 2 (EtherCAT)^Term 1 (EK1200)^Term 4 (EL3446)^I3 Channel^Apparent Power Guard Error'}
	MDP5001_342_I3_Channel_Apparent_Power_Guard_Error_EM2		AT%I*  : BOOL;
	{attribute 'TcLinkTo' := 'TIID^Device 2 (EtherCAT)^Term 1 (EK1200)^Term 4 (EL3446)^I3 Channel^Active Power Guard Warning'}
	MDP5001_342_I3_Channel_Active_Power_Guard_Warning_EM2		AT%I*  : BOOL;
	{attribute 'TcLinkTo' := 'TIID^Device 2 (EtherCAT)^Term 1 (EK1200)^Term 4 (EL3446)^I3 Channel^Active Power Guard Error'}
	MDP5001_342_I3_Channel_Active_Power_Guard_Error_EM2		AT%I*  : BOOL;
	{attribute 'TcLinkTo' := 'TIID^Device 2 (EtherCAT)^Term 1 (EK1200)^Term 4 (EL3446)^I3 Channel^Reactive Power Guard Warning'}
	MDP5001_342_I3_Channel_Reactive_Power_Guard_Warning_EM2		AT%I*  : BOOL;
	{attribute 'TcLinkTo' := 'TIID^Device 2 (EtherCAT)^Term 1 (EK1200)^Term 4 (EL3446)^I3 Channel^Reactive Power Guard Error'}
	MDP5001_342_I3_Channel_Reactive_Power_Guard_Error_EM2		AT%I*  : BOOL;
	{attribute 'TcLinkTo' := 'TIID^Device 2 (EtherCAT)^Term 1 (EK1200)^Term 4 (EL3446)^I3 Channel^DPM Inaccurate'}
	MDP5001_342_I3_Channel_DPM_Inaccurate_EM2					AT%I*  : BOOL;
	{attribute 'TcLinkTo' := 'TIID^Device 2 (EtherCAT)^Term 1 (EK1200)^Term 4 (EL3446)^I3 Channel^DPM Timeout'}
	MDP5001_342_I3_Channel_DPM_Timeout_EM2						AT%I*  : BOOL;
	{attribute 'TcLinkTo' := 'TIID^Device 2 (EtherCAT)^Term 1 (EK1200)^Term 4 (EL3446)^I3 Channel^TxPDO Toggle'}
	MDP5001_342_I3_Channel_TxPDO_Toggle_EM2						AT%I*  : BOOL;
	{attribute 'TcLinkTo' := 'TIID^Device 2 (EtherCAT)^Term 1 (EK1200)^Term 4 (EL3446)^I3 Channel^Current'}
	MDP5001_342_I3_Channel_Current_EM2							AT%I*  : REAL;
	{attribute 'TcLinkTo' := 'TIID^Device 2 (EtherCAT)^Term 1 (EK1200)^Term 4 (EL3446)^I3 Channel^Active Power'}
	MDP5001_342_I3_Channel_Active_Power_EM2						AT%I*  : REAL;
	{attribute 'TcLinkTo' := 'TIID^Device 2 (EtherCAT)^Term 1 (EK1200)^Term 4 (EL3446)^I3 Channel^Apparent Power'}
	MDP5001_342_I3_Channel_Apparent_Power_EM2					AT%I*  : REAL;
	{attribute 'TcLinkTo' := 'TIID^Device 2 (EtherCAT)^Term 1 (EK1200)^Term 4 (EL3446)^I3 Channel^Reactive Power Fundamental'}
	MDP5001_342_I3_Channel_Reactive_Power_Fundamental_EM2		AT%I*  : REAL;
	{attribute 'TcLinkTo' := 'TIID^Device 2 (EtherCAT)^Term 1 (EK1200)^Term 4 (EL3446)^I3 Channel^Active Energy'}
	MDP5001_342_I3_Channel_Active_Energy_EM2					AT%I*  : DINT;	
	{attribute 'TcLinkTo' := 'TIID^Device 2 (EtherCAT)^Term 1 (EK1200)^Term 4 (EL3446)^I4 Channel^Overcurrent'}
	MDP5001_342_I4_Channel_Overcurrent_EM2						AT%I*  : BOOL;
	{attribute 'TcLinkTo' := 'TIID^Device 2 (EtherCAT)^Term 1 (EK1200)^Term 4 (EL3446)^I4 Channel^Inaccurate Current'}
	MDP5001_342_I4_Channel_Inaccurate_Current_EM2				AT%I*  : BOOL;
	{attribute 'TcLinkTo' := 'TIID^Device 2 (EtherCAT)^Term 1 (EK1200)^Term 4 (EL3446)^I4 Channel^Current Guard Warning'}
	MDP5001_342_I4_Channel_Current_Guard_Warning_EM2			AT%I*  : BOOL;
	{attribute 'TcLinkTo' := 'TIID^Device 2 (EtherCAT)^Term 1 (EK1200)^Term 4 (EL3446)^I4 Channel^Current Guard Error'}
	MDP5001_342_I4_Channel_Current_Guard_Error_EM2				AT%I*  : BOOL;
	{attribute 'TcLinkTo' := 'TIID^Device 2 (EtherCAT)^Term 1 (EK1200)^Term 4 (EL3446)^I4 Channel^Apparent Power Guard Warning'}
	MDP5001_342_I4_Channel_Apparent_Power_Guard_Warning_EM2		AT%I*  : BOOL;
	{attribute 'TcLinkTo' := 'TIID^Device 2 (EtherCAT)^Term 1 (EK1200)^Term 4 (EL3446)^I4 Channel^Apparent Power Guard Error'}
	MDP5001_342_I4_Channel_Apparent_Power_Guard_Error_EM2		AT%I*  : BOOL;
	{attribute 'TcLinkTo' := 'TIID^Device 2 (EtherCAT)^Term 1 (EK1200)^Term 4 (EL3446)^I4 Channel^Active Power Guard Warning'}
	MDP5001_342_I4_Channel_Active_Power_Guard_Warning_EM2		AT%I*  : BOOL;
	{attribute 'TcLinkTo' := 'TIID^Device 2 (EtherCAT)^Term 1 (EK1200)^Term 4 (EL3446)^I4 Channel^Active Power Guard Error'}
	MDP5001_342_I4_Channel_Active_Power_Guard_Error_EM2			AT%I*  : BOOL;
	{attribute 'TcLinkTo' := 'TIID^Device 2 (EtherCAT)^Term 1 (EK1200)^Term 4 (EL3446)^I4 Channel^Reactive Power Guard Warning'}
	MDP5001_342_I4_Channel_Reactive_Power_Guard_Warning_EM2		AT%I*  : BOOL;
	{attribute 'TcLinkTo' := 'TIID^Device 2 (EtherCAT)^Term 1 (EK1200)^Term 4 (EL3446)^I4 Channel^Reactive Power Guard Error'}
	MDP5001_342_I4_Channel_Reactive_Power_Guard_Error_EM2		AT%I*  : BOOL;
	{attribute 'TcLinkTo' := 'TIID^Device 2 (EtherCAT)^Term 1 (EK1200)^Term 4 (EL3446)^I4 Channel^DPM Inaccurate'}
	MDP5001_342_I4_Channel_DPM_Inaccurate_EM2					AT%I*  : BOOL;
	{attribute 'TcLinkTo' := 'TIID^Device 2 (EtherCAT)^Term 1 (EK1200)^Term 4 (EL3446)^I4 Channel^DPM Timeout'}
	MDP5001_342_I4_Channel_DPM_Timeout_EM2						AT%I*  : BOOL;
	{attribute 'TcLinkTo' := 'TIID^Device 2 (EtherCAT)^Term 1 (EK1200)^Term 4 (EL3446)^I4 Channel^TxPDO Toggle'}
	MDP5001_342_I4_Channel_TxPDO_Toggle_EM2						AT%I*  : BOOL;
	{attribute 'TcLinkTo' := 'TIID^Device 2 (EtherCAT)^Term 1 (EK1200)^Term 4 (EL3446)^I4 Channel^Current'}
	MDP5001_342_I4_Channel_Current_EM2							AT%I*  : REAL;
	{attribute 'TcLinkTo' := 'TIID^Device 2 (EtherCAT)^Term 1 (EK1200)^Term 4 (EL3446)^I4 Channel^Active Power'}
	MDP5001_342_I4_Channel_Active_Power_EM2						AT%I*  : REAL;
	{attribute 'TcLinkTo' := 'TIID^Device 2 (EtherCAT)^Term 1 (EK1200)^Term 4 (EL3446)^I4 Channel^Apparent Power'}
	MDP5001_342_I4_Channel_Apparent_Power_EM2					AT%I*  : REAL;
	{attribute 'TcLinkTo' := 'TIID^Device 2 (EtherCAT)^Term 1 (EK1200)^Term 4 (EL3446)^I4 Channel^Reactive Power Fundamental'}
	MDP5001_342_I4_Channel_Reactive_Power_Fundamental_EM2		AT%I*  : REAL;
	{attribute 'TcLinkTo' := 'TIID^Device 2 (EtherCAT)^Term 1 (EK1200)^Term 4 (EL3446)^I4 Channel^Active Energy'}
	MDP5001_342_I4_Channel_Active_Energy_EM2					AT%I*  : DINT;
	{attribute 'TcLinkTo' := 'TIID^Device 2 (EtherCAT)^Term 1 (EK1200)^Term 4 (EL3446)^I5 Channel^Overcurrent'}
	MDP5001_342_I5_Channel_Overcurrent_EM2						AT%I*  : BOOL;
	{attribute 'TcLinkTo' := 'TIID^Device 2 (EtherCAT)^Term 1 (EK1200)^Term 4 (EL3446)^I5 Channel^Inaccurate Current'}
	MDP5001_342_I5_Channel_Inaccurate_Current_EM2				AT%I*  : BOOL;
	{attribute 'TcLinkTo' := 'TIID^Device 2 (EtherCAT)^Term 1 (EK1200)^Term 4 (EL3446)^I5 Channel^Current Guard Warning'}
	MDP5001_342_I5_Channel_Current_Guard_Warning_EM2			AT%I*  : BOOL;
	{attribute 'TcLinkTo' := 'TIID^Device 2 (EtherCAT)^Term 1 (EK1200)^Term 4 (EL3446)^I5 Channel^Current Guard Error'}
	MDP5001_342_I5_Channel_Current_Guard_Error_EM2				AT%I*  : BOOL;
	{attribute 'TcLinkTo' := 'TIID^Device 2 (EtherCAT)^Term 1 (EK1200)^Term 4 (EL3446)^I5 Channel^Apparent Power Guard Warning'}
	MDP5001_342_I5_Channel_Apparent_Power_Guard_Warning_EM2		AT%I*  : BOOL;
	{attribute 'TcLinkTo' := 'TIID^Device 2 (EtherCAT)^Term 1 (EK1200)^Term 4 (EL3446)^I5 Channel^Apparent Power Guard Error'}
	MDP5001_342_I5_Channel_Apparent_Power_Guard_Error_EM2		AT%I*  : BOOL;
	{attribute 'TcLinkTo' := 'TIID^Device 2 (EtherCAT)^Term 1 (EK1200)^Term 4 (EL3446)^I5 Channel^Active Power Guard Warning'}
	MDP5001_342_I5_Channel_Active_Power_Guard_Warning_EM2		AT%I*  : BOOL;
	{attribute 'TcLinkTo' := 'TIID^Device 2 (EtherCAT)^Term 1 (EK1200)^Term 4 (EL3446)^I5 Channel^Active Power Guard Error'}
	MDP5001_342_I5_Channel_Active_Power_Guard_Error_EM2			AT%I*  : BOOL;
	{attribute 'TcLinkTo' := 'TIID^Device 2 (EtherCAT)^Term 1 (EK1200)^Term 4 (EL3446)^I5 Channel^Reactive Power Guard Warning'}
	MDP5001_342_I5_Channel_Reactive_Power_Guard_Warning_EM2		AT%I*  : BOOL;
	{attribute 'TcLinkTo' := 'TIID^Device 2 (EtherCAT)^Term 1 (EK1200)^Term 4 (EL3446)^I5 Channel^Reactive Power Guard Error'}
	MDP5001_342_I5_Channel_Reactive_Power_Guard_Error_EM2		AT%I*  : BOOL;
	{attribute 'TcLinkTo' := 'TIID^Device 2 (EtherCAT)^Term 1 (EK1200)^Term 4 (EL3446)^I5 Channel^DPM Inaccurate'}
	MDP5001_342_I5_Channel_DPM_Inaccurate_EM2					AT%I*  : BOOL;
	{attribute 'TcLinkTo' := 'TIID^Device 2 (EtherCAT)^Term 1 (EK1200)^Term 4 (EL3446)^I5 Channel^DPM Timeout'}
	MDP5001_342_I5_Channel_DPM_Timeout_EM2						AT%I*  : BOOL;
	{attribute 'TcLinkTo' := 'TIID^Device 2 (EtherCAT)^Term 1 (EK1200)^Term 4 (EL3446)^I5 Channel^TxPDO Toggle'}
	MDP5001_342_I5_Channel_TxPDO_Toggle_EM2						AT%I*  : BOOL;
	{attribute 'TcLinkTo' := 'TIID^Device 2 (EtherCAT)^Term 1 (EK1200)^Term 4 (EL3446)^I5 Channel^Current'}
	MDP5001_342_I5_Channel_Current_EM2							AT%I*  : REAL;
	{attribute 'TcLinkTo' := 'TIID^Device 2 (EtherCAT)^Term 1 (EK1200)^Term 4 (EL3446)^I5 Channel^Active Power'}
	MDP5001_342_I5_Channel_Active_Power_EM2						AT%I*  : REAL;
	{attribute 'TcLinkTo' := 'TIID^Device 2 (EtherCAT)^Term 1 (EK1200)^Term 4 (EL3446)^I5 Channel^Apparent Power'}
	MDP5001_342_I5_Channel_Apparent_Power_EM2					AT%I*  : REAL;
	{attribute 'TcLinkTo' := 'TIID^Device 2 (EtherCAT)^Term 1 (EK1200)^Term 4 (EL3446)^I5 Channel^Reactive Power Fundamental'}
	MDP5001_342_I5_Channel_Reactive_Power_Fundamental_EM2		AT%I*  : REAL;
	{attribute 'TcLinkTo' := 'TIID^Device 2 (EtherCAT)^Term 1 (EK1200)^Term 4 (EL3446)^I5 Channel^Active Energy'}
	MDP5001_342_I5_Channel_Active_Energy_EM2					AT%I*  : DINT;
	{attribute 'TcLinkTo' := 'TIID^Device 2 (EtherCAT)^Term 1 (EK1200)^Term 4 (EL3446)^I6 Channel^Overcurrent'}
	MDP5001_342_I6_Channel_Overcurrent_EM2						AT%I*  : BOOL;
	{attribute 'TcLinkTo' := 'TIID^Device 2 (EtherCAT)^Term 1 (EK1200)^Term 4 (EL3446)^I6 Channel^Inaccurate Current'}
	MDP5001_342_I6_Channel_Inaccurate_Current_EM2				AT%I*  : BOOL;
	{attribute 'TcLinkTo' := 'TIID^Device 2 (EtherCAT)^Term 1 (EK1200)^Term 4 (EL3446)^I6 Channel^Current Guard Warning'}
	MDP5001_342_I6_Channel_Current_Guard_Warning_EM2			AT%I*  : BOOL;
	{attribute 'TcLinkTo' := 'TIID^Device 2 (EtherCAT)^Term 1 (EK1200)^Term 4 (EL3446)^I6 Channel^Current Guard Error'}
	MDP5001_342_I6_Channel_Current_Guard_Error_EM2				AT%I*  : BOOL;
	{attribute 'TcLinkTo' := 'TIID^Device 2 (EtherCAT)^Term 1 (EK1200)^Term 4 (EL3446)^I6 Channel^Apparent Power Guard Warning'}
	MDP5001_342_I6_Channel_Apparent_Power_Guard_Warning_EM2		AT%I*  : BOOL;
	{attribute 'TcLinkTo' := 'TIID^Device 2 (EtherCAT)^Term 1 (EK1200)^Term 4 (EL3446)^I6 Channel^Apparent Power Guard Error'}
	MDP5001_342_I6_Channel_Apparent_Power_Guard_Error_EM2		AT%I*  : BOOL;
	{attribute 'TcLinkTo' := 'TIID^Device 2 (EtherCAT)^Term 1 (EK1200)^Term 4 (EL3446)^I6 Channel^Active Power Guard Warning'}
	MDP5001_342_I6_Channel_Active_Power_Guard_Warning_EM2		AT%I*  : BOOL;
	{attribute 'TcLinkTo' := 'TIID^Device 2 (EtherCAT)^Term 1 (EK1200)^Term 4 (EL3446)^I6 Channel^Active Power Guard Error'}
	MDP5001_342_I6_Channel_Active_Power_Guard_Error_EM2			AT%I*  : BOOL;
	{attribute 'TcLinkTo' := 'TIID^Device 2 (EtherCAT)^Term 1 (EK1200)^Term 4 (EL3446)^I6 Channel^Reactive Power Guard Warning'}
	MDP5001_342_I6_Channel_Reactive_Power_Guard_Warning_EM2		AT%I*  : BOOL;
	{attribute 'TcLinkTo' := 'TIID^Device 2 (EtherCAT)^Term 1 (EK1200)^Term 4 (EL3446)^I6 Channel^Reactive Power Guard Error'}
	MDP5001_342_I6_Channel_Reactive_Power_Guard_Error_EM2		AT%I*  : BOOL;
	{attribute 'TcLinkTo' := 'TIID^Device 2 (EtherCAT)^Term 1 (EK1200)^Term 4 (EL3446)^I6 Channel^DPM Inaccurate'}
	MDP5001_342_I6_Channel_DPM_Inaccurate_EM2					AT%I*  : BOOL;
	{attribute 'TcLinkTo' := 'TIID^Device 2 (EtherCAT)^Term 1 (EK1200)^Term 4 (EL3446)^I6 Channel^DPM Timeout'}
	MDP5001_342_I6_Channel_DPM_Timeout_EM2						AT%I*  : BOOL;
	{attribute 'TcLinkTo' := 'TIID^Device 2 (EtherCAT)^Term 1 (EK1200)^Term 4 (EL3446)^I6 Channel^TxPDO Toggle'}
	MDP5001_342_I6_Channel_TxPDO_Toggle_EM2						AT%I*  : BOOL;
	{attribute 'TcLinkTo' := 'TIID^Device 2 (EtherCAT)^Term 1 (EK1200)^Term 4 (EL3446)^I6 Channel^Current'}
	MDP5001_342_I6_Channel_Current_EM2							AT%I*  : REAL;
	{attribute 'TcLinkTo' := 'TIID^Device 2 (EtherCAT)^Term 1 (EK1200)^Term 4 (EL3446)^I6 Channel^Active Power'}
	MDP5001_342_I6_Channel_Active_Power_EM2						AT%I*  : REAL;
	{attribute 'TcLinkTo' := 'TIID^Device 2 (EtherCAT)^Term 1 (EK1200)^Term 4 (EL3446)^I6 Channel^Apparent Power'}
	MDP5001_342_I6_Channel_Apparent_Power_EM2					AT%I*  : REAL;
	{attribute 'TcLinkTo' := 'TIID^Device 2 (EtherCAT)^Term 1 (EK1200)^Term 4 (EL3446)^I6 Channel^Reactive Power Fundamental'}
	MDP5001_342_I6_Channel_Reactive_Power_Fundamental_EM2		AT%I*  : REAL;
	{attribute 'TcLinkTo' := 'TIID^Device 2 (EtherCAT)^Term 1 (EK1200)^Term 4 (EL3446)^I6 Channel^Active Energy'}
	MDP5001_342_I6_Channel_Active_Energy_EM2					AT%I*  : DINT;	
	
	{attribute 'TcLinkTo' := 'TIID^Device 2 (EtherCAT)^Term 1 (EK1200)^Term 4 (EL3446)^DPM Variant Value In^TxPDO Toggle'}
	MDP5001_342_DPM_Variant_Value_In_TxPDO_Toggle_EM2			AT%I*  : BOOL;
	{attribute 'TcLinkTo' := 'TIID^Device 2 (EtherCAT)^Term 1 (EK1200)^Term 4 (EL3446)^DPM Variant Value In^Index 1 REAL'}
	MDP5001_342_DPM_Variant_Value_In_Index_1_REAL_EM2			AT%I*  : UINT;
	{attribute 'TcLinkTo' := 'TIID^Device 2 (EtherCAT)^Term 1 (EK1200)^Term 4 (EL3446)^DPM Variant Value In^Value 1 REAL'}
	MDP5001_342_DPM_Variant_Value_In_Value_1_REAL_EM2			AT%I*  : REAL;
	{attribute 'TcLinkTo' := 'TIID^Device 2 (EtherCAT)^Term 1 (EK1200)^Term 4 (EL3446)^DPM Variant Value In^Index 2 REAL'}
	MDP5001_342_DPM_Variant_Value_In_Index_2_REAL_EM2			AT%I*  : UINT;
	{attribute 'TcLinkTo' := 'TIID^Device 2 (EtherCAT)^Term 1 (EK1200)^Term 4 (EL3446)^DPM Variant Value In^Value 2 REAL'}
	MDP5001_342_DPM_Variant_Value_In_Value_2_REAL_EM2			AT%I*  : REAL;
	{attribute 'TcLinkTo' := 'TIID^Device 2 (EtherCAT)^Term 1 (EK1200)^Term 4 (EL3446)^DPM Variant Value In^Index 3 REAL'}
	MDP5001_342_DPM_Variant_Value_In_Index_3_REAL_EM2			AT%I*  : UINT;
	{attribute 'TcLinkTo' := 'TIID^Device 2 (EtherCAT)^Term 1 (EK1200)^Term 4 (EL3446)^DPM Variant Value In^Value 3 REAL'}
	MDP5001_342_DPM_Variant_Value_In_Value_3_REAL_EM2			AT%I*  : REAL;
	{attribute 'TcLinkTo' := 'TIID^Device 2 (EtherCAT)^Term 1 (EK1200)^Term 4 (EL3446)^DPM Variant Value In^Index 4 ULINT'}
	MDP5001_342_DPM_Variant_Value_In_Index_4_ULINT_EM2			AT%I*  : UINT;
	{attribute 'TcLinkTo' := 'TIID^Device 2 (EtherCAT)^Term 1 (EK1200)^Term 4 (EL3446)^DPM Variant Value In^Value 4 ULINT'}
	MDP5001_342_DPM_Variant_Value_In_Value_4_ULINT_EM2			AT%I*  : ULINT;

	{attribute 'TcLinkTo' := 'TIID^Device 2 (EtherCAT)^Term 1 (EK1200)^Term 4 (EL3446)^DPM Variant Value Out^Index 1 REAL'}
	MDP5001_342_DPM_Variant_Value_Out_Index_1_REAL_EM2	AT%Q* : UINT;
	{attribute 'TcLinkTo' := 'TIID^Device 2 (EtherCAT)^Term 1 (EK1200)^Term 4 (EL3446)^DPM Variant Value Out^Index 2 REAL'}
	MDP5001_342_DPM_Variant_Value_Out_Index_2_REAL_EM2	AT%Q* : UINT;
	{attribute 'TcLinkTo' := 'TIID^Device 2 (EtherCAT)^Term 1 (EK1200)^Term 4 (EL3446)^DPM Variant Value Out^Index 3 REAL'}
	MDP5001_342_DPM_Variant_Value_Out_Index_3_REAL_EM2	AT%Q* : UINT;
	{attribute 'TcLinkTo' := 'TIID^Device 2 (EtherCAT)^Term 1 (EK1200)^Term 4 (EL3446)^DPM Variant Value Out^Index 4 ULINT'}
	MDP5001_342_DPM_Variant_Value_Out_Index_4_ULINT_EM2	AT%Q* : UINT;
	{attribute 'TcLinkTo' := 'TIID^Device 2 (EtherCAT)^Term 1 (EK1200)^Term 4 (EL3446)^DPM Data^Data 1'}
	MDP5001_342_DPM_Data_Data_1_EM2						AT%Q* : UDINT;
	{attribute 'TcLinkTo' := 'TIID^Device 2 (EtherCAT)^Term 1 (EK1200)^Term 4 (EL3446)^DPM Data^Data 2'}
	MDP5001_342_DPM_Data_Data_2_EM2						AT%Q* : UDINT;
	{attribute 'TcLinkTo' := 'TIID^Device 2 (EtherCAT)^Term 1 (EK1200)^Term 4 (EL3446)^DPM Data^Data 3'}
	MDP5001_342_DPM_Data_Data_3_EM2						AT%Q* : UDINT;
	{attribute 'TcLinkTo' := 'TIID^Device 2 (EtherCAT)^Term 1 (EK1200)^Term 4 (EL3446)^DPM Data^Data 4'}
	MDP5001_342_DPM_Data_Data_4_EM2						AT%Q* : UDINT;
	{attribute 'TcLinkTo' := 'TIID^Device 2 (EtherCAT)^Term 1 (EK1200)^Term 4 (EL3446)^DPM Data^Data 5'}
	MDP5001_342_DPM_Data_Data_5_EM2						AT%Q* : UDINT;
	{attribute 'TcLinkTo' := 'TIID^Device 2 (EtherCAT)^Term 1 (EK1200)^Term 4 (EL3446)^DPM Data^Data 6'}
	MDP5001_342_DPM_Data_Data_6_EM2						AT%Q* : UDINT;
	{attribute 'TcLinkTo' := 'TIID^Device 2 (EtherCAT)^Term 1 (EK1200)^Term 4 (EL3446)^DPM Data^Data 7'}
	MDP5001_342_DPM_Data_Data_7_EM2						AT%Q* : UDINT;
	{attribute 'TcLinkTo' := 'TIID^Device 2 (EtherCAT)^Term 1 (EK1200)^Term 4 (EL3446)^DPM Data^Data 8'}
	MDP5001_342_DPM_Data_Data_8_EM2						AT%Q* : UDINT;
	{attribute 'TcLinkTo' := 'TIID^Device 2 (EtherCAT)^Term 1 (EK1200)^Term 4 (EL3446)^DPM Data^Data 9'}
	MDP5001_342_DPM_Data_Data_9_EM2						AT%Q* : UDINT;
	{attribute 'TcLinkTo' := 'TIID^Device 2 (EtherCAT)^Term 1 (EK1200)^Term 4 (EL3446)^DPM Data^Data 10'}
	MDP5001_342_DPM_Data_Data_10_EM2					AT%Q* : UDINT;
	{attribute 'TcLinkTo' := 'TIID^Device 2 (EtherCAT)^Term 1 (EK1200)^Term 4 (EL3446)^DPM Data^Data 11'}
	MDP5001_342_DPM_Data_Data_11_EM2					AT%Q* : UDINT;
	{attribute 'TcLinkTo' := 'TIID^Device 2 (EtherCAT)^Term 1 (EK1200)^Term 4 (EL3446)^DPM Data^Data 12'}
	MDP5001_342_DPM_Data_Data_12_EM2					AT%Q* : UDINT;
	{attribute 'TcLinkTo' := 'TIID^Device 2 (EtherCAT)^Term 1 (EK1200)^Term 4 (EL3446)^DPM Data^Data 13'}
	MDP5001_342_DPM_Data_Data_13_EM2					AT%Q* : UDINT;
	{attribute 'TcLinkTo' := 'TIID^Device 2 (EtherCAT)^Term 1 (EK1200)^Term 4 (EL3446)^DPM Data^Data 14'}
	MDP5001_342_DPM_Data_Data_14_EM2					AT%Q* : UDINT;
	{attribute 'TcLinkTo' := 'TIID^Device 2 (EtherCAT)^Term 1 (EK1200)^Term 4 (EL3446)^DPM Data^Data 15'}
	MDP5001_342_DPM_Data_Data_15_EM2					AT%Q* : UDINT;
	{attribute 'TcLinkTo' := 'TIID^Device 2 (EtherCAT)^Term 1 (EK1200)^Term 4 (EL3446)^DPM Data^Data 16'}
	MDP5001_342_DPM_Data_Data_16_EM2					AT%Q* : UDINT;
	{attribute 'TcLinkTo' := 'TIID^Device 2 (EtherCAT)^Term 1 (EK1200)^Term 4 (EL3446)^DPM Data^Data 17'}
	MDP5001_342_DPM_Data_Data_17_EM2					AT%Q* : UDINT;
	{attribute 'TcLinkTo' := 'TIID^Device 2 (EtherCAT)^Term 1 (EK1200)^Term 4 (EL3446)^DPM Data^Data 18'}
	MDP5001_342_DPM_Data_Data_18_EM2					AT%Q* : UDINT;
	{attribute 'TcLinkTo' := 'TIID^Device 2 (EtherCAT)^Term 1 (EK1200)^Term 4 (EL3446)^DPM Data^Data 19'}
	MDP5001_342_DPM_Data_Data_19_EM2					AT%Q* : UDINT;
	{attribute 'TcLinkTo' := 'TIID^Device 2 (EtherCAT)^Term 1 (EK1200)^Term 4 (EL3446)^DPM Data^Data 20'}
	MDP5001_342_DPM_Data_Data_20_EM2					AT%Q* : UDINT;

